ABB RobotStudio station: change_path.rspag

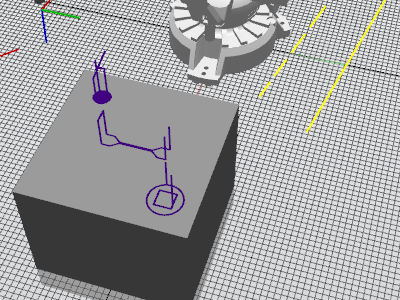
--- station ---
Station themal simulation (saved by RobotStudio 25.1.11133.0)
Controller IRB2600_12_185
  mechanical unit ROB_1: IRB2600_12_185__02, 6 joints, base frame (0, 0, 0) mm
Layout (positions relative to the parent item):
  - IRB2600_12_185__02 [mechanism, from %ABB.RobotStudio.Models.IRB2600%\IRB2600_12_185_G_02.rslib] at (0, 0, 0) mm; joint values [0, 0, 0, 0, 0.5236, 0] (rad or m)
  - AW_Gun_PSF_25 [mechanism, from %ABB.RobotStudio.Models.ArcWelding%\AW_Gun_PSF_25.rslib] at (1018.61, 0, 1417.5) mm, rotated rx 180 ry 60 rz 180 deg
  - Part_1 [part] at (100, 0, -100) mm, size 500 x 500 x 500 mm
Attachment: AW_Gun_PSF_25 is attached to IRB2600_12_185__02 / Link6

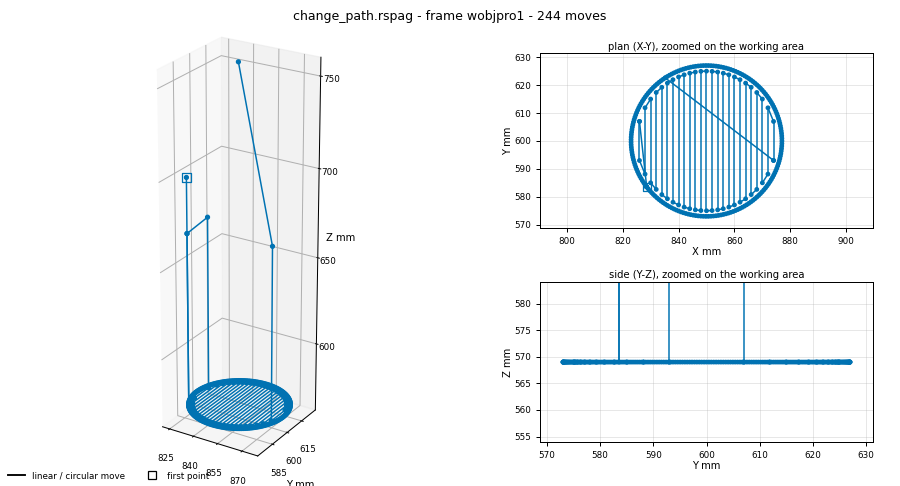
[picture p0: tool path of change_path.rspag in frame wobjpro1, 244 of 529 moves have a stored position in this frame; points joined in program order, loops and branches not executed]
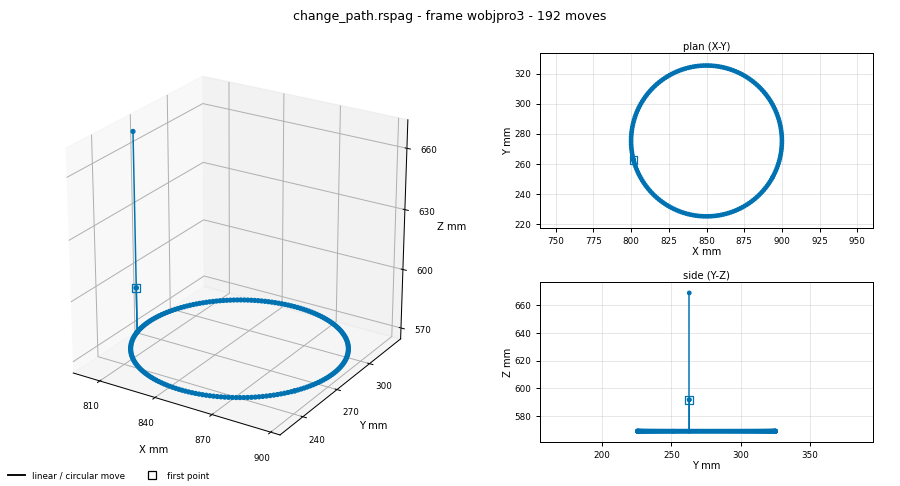
[picture p1: tool path of change_path.rspag in frame wobjpro3, 192 of 529 moves have a stored position in this frame; points joined in program order, loops and branches not executed]
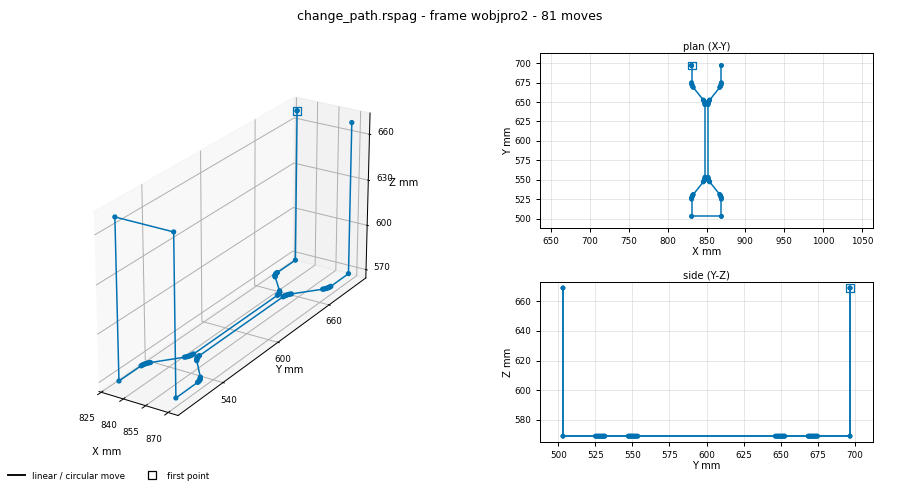
[picture p2: tool path of change_path.rspag in frame wobjpro2, 81 of 529 moves have a stored position in this frame; points joined in program order, loops and branches not executed]
--- Controller Data/IRB2600_12_185/RAPID/TASK1/PROGMOD/CalibData.mod ---
MODULE CalibData
    PERS tooldata AW_Gun:=[TRUE,[[119.5,0,352],[0.890213743,0,0.455543074,0]],[1,[0,0,100],[1,0,0,0],0,0,0]];
    PERS tooldata tFronius:=[TRUE,[[119.5,0,352],[0.890213743,0,0.455543074,0]],[1,[0,0,100],[1,0,0,0],0,0,0]];
     TASK PERS wobjdata wobjpro1:=[FALSE,TRUE,"",[[-52.352266096,-751.940840166,-168.793042727],[1,0,0,0]],[[0,0,0.0541992],[1,0,0,0]]];
  TASK PERS wobjdata wobjpro2:=[FALSE,TRUE,"",[[101.173073889,-585.583883348,-168],[1,0,0,0]],[[0,0,-0.0836792],[1,0,0,0]]];
  TASK PERS wobjdata wobjpro3:=[FALSE,TRUE,"",[[251.773303947,-119.398296432,-164.096623534],[1,0,0,0]],[[0,0,-4.67993],[1,0,0,0]]];
   TASK PERS wobjdata wobjpro4:=[FALSE,TRUE,"",[[250.933389795,-444.202986893,-163.664818503],[1,0,0,0]],[[0,0,-5.12018],[1,0,0,0]]];
  TASK PERS wobjdata wobjcam:=[FALSE,TRUE,"",[[1100,380,580],[1,0,0,0]],[[0,0,0],[1,0,0,0]]];
  TASK PERS wobjdata dedicate_wobj:=[FALSE,TRUE,"",[[1003,385,578.53],[1,0,0,0]],[[0,0,11.1832],[1,0,0,0]]];


PERS tooldata Processhead1 := [TRUE,[[-1.72,-0.76,490.02],[-0.01344,-0.95371,-0.07753,0.29025]],[3,[1,0,300],[1,0,0,0],0,0,0]];


!! ************************************************************
!! Toolpath ID: 1724238657_MX3D8v7kg | MX3D
!! Chunk ID: 0 [1/1]
!! Robot: hv_waam cell
!! Filename: MX3D_20240821_151151.mod
!! Project name: MX3D
!! Created on 2024-08-21 15:11:51.971757
!! ************************************************************

!! Delays for 2mm layer strategy (Single Wall Contour):
VAR num delayClosedStart_0  := 0.05;
VAR num delayClosedStop_0   := 0.05;
VAR num delayOpenStart_0    := 0.25;
VAR num delayOpenStop_0     := 0.1;


!! Delays for 2.6 mm layer strategy (Single Wall Contour):
VAR num delayClosedStart_1  := 0.05;
VAR num delayClosedStop_1   := 0.05;
VAR num delayOpenStart_1    := 0.1;
VAR num delayOpenStop_1     := 0.1;

VAR num delayOverhang       := 0;

!! Print and approach speeds
VAR speeddata printSpeed := [12, 500.0, 10.0, 10.0];
VAR speeddata moveSpeed := [800.0, 500.0, 300.0, 60.0];

!! Welding and process parameters
VAR bool useTempSensor    := TRUE;

VAR num wTime_25 := 25;
 CONST robtarget p30:=[[-49.36,-18.80,327.48],[0.761522,-0.0130271,0.0123584,0.647891],[0,1,-2,0],[9E+09,9E+09,9E+09,9E+09,9E+09,9E+09]];


VAR num wTime_5 := 5;

 !!PERS tooldata bendedTool:=[TRUE,[[-1.728,-0.7687,490.03],[0.0775305,-0.290248,-0.0134406,-0.953711]],[10,[85,0,65],[1,0,0,0],0.01,0.01,0.01]];
 PERS tooldata bendedTool:=[TRUE,[[119.5,0,352],[0.890213743,0,0.455543074,0]],[1,[0,0,100],[1,0,0,0],0,0,0]];
    TASK PERS wobjdata wobjWelding:=[FALSE,TRUE,"",[[700,-250,400],[1,0,0,0]],[[0,0,0],[1,0,0,0]]];
ENDMODULE

--- Controller Data/IRB2600_12_185/RAPID/TASK1/PROGMOD/Module1.mod ---
MODULE Module1
        CONST robtarget Target_10:=[[100,100,50],[0,0,1,0],[-1,1,-2,0],[9E+09,9E+09,9E+09,9E+09,9E+09,9E+09]];
    CONST robtarget Target_20:=[[100,400,50],[0,0,1,0],[0,2,-3,0],[9E+09,9E+09,9E+09,9E+09,9E+09,9E+09]];
    CONST robtarget Target_30:=[[400,400,50],[0,0,1,0],[0,2,-3,0],[9E+09,9E+09,9E+09,9E+09,9E+09,9E+09]];
    CONST robtarget Target_40:=[[400,100,50],[0,0,1,0],[-1,1,-2,0],[9E+09,9E+09,9E+09,9E+09,9E+09,9E+09]];
    CONST robtarget Target_50:=[[250,250,0],[0,0,1,0],[0,1,-2,0],[9E+09,9E+09,9E+09,9E+09,9E+09,9E+09]];
    CONST robtarget Target_10_1:=[[120,80,0],[0,0,1,0],[-1,1,-2,0],[9E+09,9E+09,9E+09,9E+09,9E+09,9E+09]];
    CONST robtarget Target_10_2:=[[80,80,0],[0,0,1,0],[-1,1,-2,0],[9E+09,9E+09,9E+09,9E+09,9E+09,9E+09]];
    CONST robtarget Target_10_3:=[[80,120,0],[0,0,1,0],[-1,1,-2,0],[9E+09,9E+09,9E+09,9E+09,9E+09,9E+09]];
    CONST robtarget Target_10_4:=[[120,120,0],[0,0,1,0],[-1,1,-2,0],[9E+09,9E+09,9E+09,9E+09,9E+09,9E+09]];
    CONST robtarget Target_20_1:=[[120,380,0],[0,0,1,0],[0,2,-3,0],[9E+09,9E+09,9E+09,9E+09,9E+09,9E+09]];
    CONST robtarget Target_20_2:=[[80,380,0],[0,0,1,0],[0,2,-3,0],[9E+09,9E+09,9E+09,9E+09,9E+09,9E+09]];
    CONST robtarget Target_20_3:=[[80,420,0],[0,0,1,0],[0,2,-3,0],[9E+09,9E+09,9E+09,9E+09,9E+09,9E+09]];
    CONST robtarget Target_20_4:=[[120,420,0],[0,0,1,0],[0,2,-3,0],[9E+09,9E+09,9E+09,9E+09,9E+09,9E+09]];
    CONST robtarget Target_30_1:=[[420,380,0],[0,0,1,0],[0,2,-3,0],[9E+09,9E+09,9E+09,9E+09,9E+09,9E+09]];
    CONST robtarget Target_30_2:=[[380,380,0],[0,0,1,0],[0,2,-3,0],[9E+09,9E+09,9E+09,9E+09,9E+09,9E+09]];
    CONST robtarget Target_30_3:=[[380,420,0],[0,0,1,0],[0,2,-3,0],[9E+09,9E+09,9E+09,9E+09,9E+09,9E+09]];
    CONST robtarget Target_30_4:=[[420,420,0],[0,0,1,0],[0,2,-3,0],[9E+09,9E+09,9E+09,9E+09,9E+09,9E+09]];
    CONST robtarget Target_40_1:=[[420,80,0],[0,0,1,0],[-1,1,-2,0],[9E+09,9E+09,9E+09,9E+09,9E+09,9E+09]];
    CONST robtarget Target_40_2:=[[380,80,0],[0,0,1,0],[-1,1,-2,0],[9E+09,9E+09,9E+09,9E+09,9E+09,9E+09]];
    CONST robtarget Target_40_3:=[[380,120,0],[0,0,1,0],[-1,1,-2,0],[9E+09,9E+09,9E+09,9E+09,9E+09,9E+09]];
    CONST robtarget Target_40_4:=[[420,120,0],[0,0,1,0],[-1,1,-2,0],[9E+09,9E+09,9E+09,9E+09,9E+09,9E+09]];
    VAR num interpassTemp;
    VAR num emissivity;
    VAR num numtemp;


!***********************************************************
    !
    ! Module:  Module1
    !
    ! Description:
    !   <Insert description here>
    !
    ! Author: xizh0002
    !
    ! Version: 1.0
    !
    !***********************************************************


    !***********************************************************
    !
    ! Procedure main
    !
    !   This is the entry point of your program
    !
    !***********************************************************
    PROC main()
        tempmeas;
    ENDPROC

    PROC tempmeas()
        r_cutwire;
    	MoveJ [[-130.39,-18.86,150.5],[0.0697509,0.000014922,-0.000044012,-0.997564],[0,-1,0,0],[9E+09,9E+09,9E+09,9E+09,9E+09,9E+09]],v500,z50,bendedTool\WObj:=wobjcam;
    	MoveJ [[31.69,367.16,1210],[0.276174,0.456891,0.112412,-0.838058],[0,0,-1,0],[9E+09,9E+09,9E+09,9E+09,9E+09,9E+09]],v800,z50,bendedTool\WObj:=wobjcam;
        tpreadfk reg1,"What to print?", "dia100","square","fork","solid","SKIP";
        MoveL [[-8.44,117.89,200],[0.0697498,-0.00001779,-0.00000352,-0.997564],[0,-1,0,0],[9E+09,9E+09,9E+09,9E+09,9E+09,9E+09]],v500,z50,bendedTool\WObj:=wobjcam;
        IF reg1=1 THEN
            dia100;
        ENDIF

        IF reg1=2 THEN
            square;
        ENDIF

        IF reg1=3 THEN
            gaffel;
        ENDIF

        IF reg1=4 THEN
            solid;
        ENDIF
    ENDPROC


PROC solid()
VAR robtarget touchpoint:=[[824.662,609.333,565],[0.000000,0.997564,0.069756,0.000000],[0,-1,0,0],[9E9,9E9,9E9,9E9,9E9,9E9]];
interpassTemp := 200.0;
emissivity := 0.992;
MoveL [[828.586,583.552,700],[0,0.997564,0.069756,0],[0,-1,0,0],[9E+09,9E+09,9E+09,9E+09,9E+09,9E+09]],moveSpeed,z0,bendedTool\WObj:=wobjpro1;
serch_height 0,0,touchpoint,numtemp;
!(num ofx, num ofy, robtarget target, inout num zval)
wobjpro1.oframe.trans.z:=numtemp-569.010;



MoveL [[828.586,583.552,669],[0,0.997564,0.069756,0],[0,-1,0,0],[9E+09,9E+09,9E+09,9E+09,9E+09,9E+09]],moveSpeed,z0,bendedTool\WObj:=wobjpro1;
MoveL [[828.586,583.552,569.01],[0,0.997564,0.069756,0],[0,-1,0,0],[9E+09,9E+09,9E+09,9E+09,9E+09,9E+09]],moveSpeed,fine,bendedTool\WObj:=wobjpro1;

startcontinuousweld; !layer  \delay:=delayClosedStart_0 \weldingProgram:=3 \weldId:="0000-0000-0000-0002";
TPWrite "[0.5%] PRT0 LYR0 TRK0 (700.0mm)";
MoveL [[828.048,584.277,569.01],[0,0.997564,0.069756,0],[0,-1,0,0],[9E+09,9E+09,9E+09,9E+09,9E+09,9E+09]],printSpeed,z0,bendedTool\WObj:=wobjpro1;
MoveL [[827.532,585.023,569.01],[0,0.997564,0.069756,0],[0,-1,0,0],[9E+09,9E+09,9E+09,9E+09,9E+09,9E+09]],printSpeed,z0,bendedTool\WObj:=wobjpro1;
MoveL [[827.042,585.786,569.01],[0,0.997564,0.069756,0],[0,-1,0,0],[9E+09,9E+09,9E+09,9E+09,9E+09,9E+09]],printSpeed,z0,bendedTool\WObj:=wobjpro1;
MoveL [[826.575,586.569,569.01],[0,0.997564,0.069756,0],[0,-1,0,0],[9E+09,9E+09,9E+09,9E+09,9E+09,9E+09]],printSpeed,z0,bendedTool\WObj:=wobjpro1;
MoveL [[826.139,587.36,569.01],[0,0.997564,0.069756,0],[0,-1,0,0],[9E+09,9E+09,9E+09,9E+09,9E+09,9E+09]],printSpeed,z0,bendedTool\WObj:=wobjpro1;
MoveL [[825.728,588.168,569.01],[0,0.997564,0.069756,0],[0,-1,0,0],[9E+09,9E+09,9E+09,9E+09,9E+09,9E+09]],printSpeed,z0,bendedTool\WObj:=wobjpro1;
MoveL [[825.344,588.99,569.01],[0,0.997564,0.069756,0],[0,-1,0,0],[9E+09,9E+09,9E+09,9E+09,9E+09,9E+09]],printSpeed,z0,bendedTool\WObj:=wobjpro1;
MoveL [[824.988,589.825,569.01],[0,0.997564,0.069756,0],[0,-1,0,0],[9E+09,9E+09,9E+09,9E+09,9E+09,9E+09]],printSpeed,z0,bendedTool\WObj:=wobjpro1;
MoveL [[824.661,590.671,569.01],[0,0.997564,0.069756,0],[0,-1,0,0],[9E+09,9E+09,9E+09,9E+09,9E+09,9E+09]],printSpeed,z0,bendedTool\WObj:=wobjpro1;
MoveL [[824.362,591.527,569.01],[0,0.997564,0.069756,0],[0,-1,0,0],[9E+09,9E+09,9E+09,9E+09,9E+09,9E+09]],printSpeed,z0,bendedTool\WObj:=wobjpro1;
MoveL [[824.091,592.393,569.01],[0,0.997564,0.069756,0],[0,-1,0,0],[9E+09,9E+09,9E+09,9E+09,9E+09,9E+09]],printSpeed,z0,bendedTool\WObj:=wobjpro1;
MoveL [[823.849,593.272,569.01],[0,0.997564,0.069756,0],[0,-1,0,0],[9E+09,9E+09,9E+09,9E+09,9E+09,9E+09]],printSpeed,z0,bendedTool\WObj:=wobjpro1;
MoveL [[823.639,594.15,569.01],[0,0.997564,0.069756,0],[0,-1,0,0],[9E+09,9E+09,9E+09,9E+09,9E+09,9E+09]],printSpeed,z0,bendedTool\WObj:=wobjpro1;
MoveL [[823.457,595.039,569.01],[0,0.997564,0.069756,0],[0,-1,0,0],[9E+09,9E+09,9E+09,9E+09,9E+09,9E+09]],printSpeed,z0,bendedTool\WObj:=wobjpro1;
MoveL [[823.306,595.933,569.01],[0,0.997564,0.069756,0],[0,-1,0,0],[9E+09,9E+09,9E+09,9E+09,9E+09,9E+09]],printSpeed,z0,bendedTool\WObj:=wobjpro1;
MoveL [[823.184,596.836,569.01],[0,0.997564,0.069756,0],[0,-1,0,0],[9E+09,9E+09,9E+09,9E+09,9E+09,9E+09]],printSpeed,z0,bendedTool\WObj:=wobjpro1;
MoveL [[823.093,597.735,569.01],[0,0.997564,0.069756,0],[0,-1,0,0],[9E+09,9E+09,9E+09,9E+09,9E+09,9E+09]],printSpeed,z0,bendedTool\WObj:=wobjpro1;
MoveL [[823.032,598.644,569.01],[0,0.997564,0.069756,0],[0,-1,0,0],[9E+09,9E+09,9E+09,9E+09,9E+09,9E+09]],printSpeed,z0,bendedTool\WObj:=wobjpro1;
MoveL [[823.002,599.551,569.01],[0,0.997564,0.069756,0],[0,-1,0,0],[9E+09,9E+09,9E+09,9E+09,9E+09,9E+09]],printSpeed,z0,bendedTool\WObj:=wobjpro1;
MoveL [[823.002,600.454,569.01],[0,0.997564,0.069756,0],[0,-1,0,0],[9E+09,9E+09,9E+09,9E+09,9E+09,9E+09]],printSpeed,z0,bendedTool\WObj:=wobjpro1;
MoveL [[823.032,601.36,569.01],[0,0.997564,0.069756,0],[0,-1,0,0],[9E+09,9E+09,9E+09,9E+09,9E+09,9E+09]],printSpeed,z0,bendedTool\WObj:=wobjpro1;
MoveL [[823.093,602.265,569.01],[0,0.997564,0.069756,0],[0,-1,0,0],[9E+09,9E+09,9E+09,9E+09,9E+09,9E+09]],printSpeed,z0,bendedTool\WObj:=wobjpro1;
MoveL [[823.184,603.168,569.01],[0,0.997564,0.069756,0],[0,-1,0,0],[9E+09,9E+09,9E+09,9E+09,9E+09,9E+09]],printSpeed,z0,bendedTool\WObj:=wobjpro1;
MoveL [[823.306,604.071,569.01],[0,0.997564,0.069756,0],[0,-1,0,0],[9E+09,9E+09,9E+09,9E+09,9E+09,9E+09]],printSpeed,z0,bendedTool\WObj:=wobjpro1;
MoveL [[823.457,604.961,569.01],[0,0.997564,0.069756,0],[0,-1,0,0],[9E+09,9E+09,9E+09,9E+09,9E+09,9E+09]],printSpeed,z0,bendedTool\WObj:=wobjpro1;
MoveL [[823.639,605.85,569.01],[0,0.997564,0.069756,0],[0,-1,0,0],[9E+09,9E+09,9E+09,9E+09,9E+09,9E+09]],printSpeed,z0,bendedTool\WObj:=wobjpro1;
MoveL [[823.85,606.732,569.01],[0,0.997564,0.069756,0],[0,-1,0,0],[9E+09,9E+09,9E+09,9E+09,9E+09,9E+09]],printSpeed,z0,bendedTool\WObj:=wobjpro1;
MoveL [[824.091,607.607,569.01],[0,0.997564,0.069756,0],[0,-1,0,0],[9E+09,9E+09,9E+09,9E+09,9E+09,9E+09]],printSpeed,z0,bendedTool\WObj:=wobjpro1;
MoveL [[824.363,608.477,569.01],[0,0.997564,0.069756,0],[0,-1,0,0],[9E+09,9E+09,9E+09,9E+09,9E+09,9E+09]],printSpeed,z0,bendedTool\WObj:=wobjpro1;
MoveL [[824.662,609.333,569.01],[0,0.997564,0.069756,0],[0,-1,0,0],[9E+09,9E+09,9E+09,9E+09,9E+09,9E+09]],printSpeed,z0,bendedTool\WObj:=wobjpro1;
MoveL [[824.988,610.175,569.01],[0,0.997564,0.069756,0],[0,-1,0,0],[9E+09,9E+09,9E+09,9E+09,9E+09,9E+09]],printSpeed,z0,bendedTool\WObj:=wobjpro1;
MoveL [[825.344,611.01,569.01],[0,0.997564,0.069756,0],[0,-1,0,0],[9E+09,9E+09,9E+09,9E+09,9E+09,9E+09]],printSpeed,z0,bendedTool\WObj:=wobjpro1;
MoveL [[825.73,611.836,569.01],[0,0.997564,0.069756,0],[0,-1,0,0],[9E+09,9E+09,9E+09,9E+09,9E+09,9E+09]],printSpeed,z0,bendedTool\WObj:=wobjpro1;
MoveL [[826.139,612.64,569.01],[0,0.997564,0.069756,0],[0,-1,0,0],[9E+09,9E+09,9E+09,9E+09,9E+09,9E+09]],printSpeed,z0,bendedTool\WObj:=wobjpro1;
MoveL [[826.577,613.435,569.01],[0,0.997564,0.069756,0],[0,-1,0,0],[9E+09,9E+09,9E+09,9E+09,9E+09,9E+09]],printSpeed,z0,bendedTool\WObj:=wobjpro1;
MoveL [[827.044,614.218,569.01],[0,0.997564,0.069756,0],[0,-1,0,0],[9E+09,9E+09,9E+09,9E+09,9E+09,9E+09]],printSpeed,z0,bendedTool\WObj:=wobjpro1;
MoveL [[827.535,614.981,569.01],[0,0.997564,0.069756,0],[0,-1,0,0],[9E+09,9E+09,9E+09,9E+09,9E+09,9E+09]],printSpeed,z0,bendedTool\WObj:=wobjpro1;
MoveL [[828.048,615.723,569.01],[0,0.997564,0.069756,0],[0,-1,0,0],[9E+09,9E+09,9E+09,9E+09,9E+09,9E+09]],printSpeed,z0,bendedTool\WObj:=wobjpro1;
MoveL [[828.589,616.452,569.01],[0,0.997564,0.069756,0],[0,-1,0,0],[9E+09,9E+09,9E+09,9E+09,9E+09,9E+09]],printSpeed,z0,bendedTool\WObj:=wobjpro1;
MoveL [[829.156,617.165,569.01],[0,0.997564,0.069756,0],[0,-1,0,0],[9E+09,9E+09,9E+09,9E+09,9E+09,9E+09]],printSpeed,z0,bendedTool\WObj:=wobjpro1;
MoveL [[829.742,617.852,569.01],[0,0.997564,0.069756,0],[0,-1,0,0],[9E+09,9E+09,9E+09,9E+09,9E+09,9E+09]],printSpeed,z0,bendedTool\WObj:=wobjpro1;
MoveL [[830.356,618.526,569.01],[0,0.997564,0.069756,0],[0,-1,0,0],[9E+09,9E+09,9E+09,9E+09,9E+09,9E+09]],printSpeed,z0,bendedTool\WObj:=wobjpro1;
MoveL [[830.986,619.172,569.01],[0,0.997564,0.069756,0],[0,-1,0,0],[9E+09,9E+09,9E+09,9E+09,9E+09,9E+09]],printSpeed,z0,bendedTool\WObj:=wobjpro1;
MoveL [[831.641,619.8,569.01],[0,0.997564,0.069756,0],[0,-1,0,0],[9E+09,9E+09,9E+09,9E+09,9E+09,9E+09]],printSpeed,z0,bendedTool\WObj:=wobjpro1;
MoveL [[832.317,620.405,569.01],[0,0.997564,0.069756,0],[0,-1,0,0],[9E+09,9E+09,9E+09,9E+09,9E+09,9E+09]],printSpeed,z0,bendedTool\WObj:=wobjpro1;
MoveL [[833.012,620.988,569.01],[0,0.997564,0.069756,0],[0,-1,0,0],[9E+09,9E+09,9E+09,9E+09,9E+09,9E+09]],printSpeed,z0,bendedTool\WObj:=wobjpro1;
MoveL [[833.727,621.547,569.01],[0,0.997564,0.069756,0],[0,-1,0,0],[9E+09,9E+09,9E+09,9E+09,9E+09,9E+09]],printSpeed,z0,bendedTool\WObj:=wobjpro1;
MoveL [[834.46,622.081,569.01],[0,0.997564,0.069756,0],[0,-1,0,0],[9E+09,9E+09,9E+09,9E+09,9E+09,9E+09]],printSpeed,z0,bendedTool\WObj:=wobjpro1;
MoveL [[835.21,622.591,569.01],[0,0.997564,0.069756,0],[0,-1,0,0],[9E+09,9E+09,9E+09,9E+09,9E+09,9E+09]],printSpeed,z0,bendedTool\WObj:=wobjpro1;
MoveL [[835.978,623.075,569.01],[0,0.997564,0.069756,0],[0,-1,0,0],[9E+09,9E+09,9E+09,9E+09,9E+09,9E+09]],printSpeed,z0,bendedTool\WObj:=wobjpro1;
MoveL [[836.761,623.533,569.01],[0,0.997564,0.069756,0],[0,-1,0,0],[9E+09,9E+09,9E+09,9E+09,9E+09,9E+09]],printSpeed,z0,bendedTool\WObj:=wobjpro1;
MoveL [[837.563,623.966,569.01],[0,0.997564,0.069756,0],[0,-1,0,0],[9E+09,9E+09,9E+09,9E+09,9E+09,9E+09]],printSpeed,z0,bendedTool\WObj:=wobjpro1;
MoveL [[838.371,624.368,569.01],[0,0.997564,0.069756,0],[0,-1,0,0],[9E+09,9E+09,9E+09,9E+09,9E+09,9E+09]],printSpeed,z0,bendedTool\WObj:=wobjpro1;
MoveL [[839.196,624.745,569.01],[0,0.997564,0.069756,0],[0,-1,0,0],[9E+09,9E+09,9E+09,9E+09,9E+09,9E+09]],printSpeed,z0,bendedTool\WObj:=wobjpro1;
MoveL [[840.033,625.094,569.01],[0,0.997564,0.069756,0],[0,-1,0,0],[9E+09,9E+09,9E+09,9E+09,9E+09,9E+09]],printSpeed,z0,bendedTool\WObj:=wobjpro1;
MoveL [[840.886,625.416,569.01],[0,0.997564,0.069756,0],[0,-1,0,0],[9E+09,9E+09,9E+09,9E+09,9E+09,9E+09]],printSpeed,z0,bendedTool\WObj:=wobjpro1;
MoveL [[841.741,625.707,569.01],[0,0.997564,0.069756,0],[0,-1,0,0],[9E+09,9E+09,9E+09,9E+09,9E+09,9E+09]],printSpeed,z0,bendedTool\WObj:=wobjpro1;
MoveL [[842.609,625.97,569.01],[0,0.997564,0.069756,0],[0,-1,0,0],[9E+09,9E+09,9E+09,9E+09,9E+09,9E+09]],printSpeed,z0,bendedTool\WObj:=wobjpro1;
MoveL [[843.49,626.204,569.01],[0,0.997564,0.069756,0],[0,-1,0,0],[9E+09,9E+09,9E+09,9E+09,9E+09,9E+09]],printSpeed,z0,bendedTool\WObj:=wobjpro1;
MoveL [[844.37,626.407,569.01],[0,0.997564,0.069756,0],[0,-1,0,0],[9E+09,9E+09,9E+09,9E+09,9E+09,9E+09]],printSpeed,z0,bendedTool\WObj:=wobjpro1;
MoveL [[845.264,626.582,569.01],[0,0.997564,0.069756,0],[0,-1,0,0],[9E+09,9E+09,9E+09,9E+09,9E+09,9E+09]],printSpeed,z0,bendedTool\WObj:=wobjpro1;
MoveL [[846.155,626.725,569.01],[0,0.997564,0.069756,0],[0,-1,0,0],[9E+09,9E+09,9E+09,9E+09,9E+09,9E+09]],printSpeed,z0,bendedTool\WObj:=wobjpro1;
MoveL [[847.055,626.839,569.01],[0,0.997564,0.069756,0],[0,-1,0,0],[9E+09,9E+09,9E+09,9E+09,9E+09,9E+09]],printSpeed,z0,bendedTool\WObj:=wobjpro1;
MoveL [[847.959,626.923,569.01],[0,0.997564,0.069756,0],[0,-1,0,0],[9E+09,9E+09,9E+09,9E+09,9E+09,9E+09]],printSpeed,z0,bendedTool\WObj:=wobjpro1;
MoveL [[848.864,626.976,569.01],[0,0.997564,0.069756,0],[0,-1,0,0],[9E+09,9E+09,9E+09,9E+09,9E+09,9E+09]],printSpeed,z0,bendedTool\WObj:=wobjpro1;
MoveL [[849.776,626.999,569.01],[0,0.997564,0.069756,0],[0,-1,0,0],[9E+09,9E+09,9E+09,9E+09,9E+09,9E+09]],printSpeed,z0,bendedTool\WObj:=wobjpro1;
MoveL [[850.679,626.992,569.01],[0,0.997564,0.069756,0],[0,-1,0,0],[9E+09,9E+09,9E+09,9E+09,9E+09,9E+09]],printSpeed,z0,bendedTool\WObj:=wobjpro1;
MoveL [[851.589,626.953,569.01],[0,0.997564,0.069756,0],[0,-1,0,0],[9E+09,9E+09,9E+09,9E+09,9E+09,9E+09]],printSpeed,z0,bendedTool\WObj:=wobjpro1;
MoveL [[852.489,626.885,569.01],[0,0.997564,0.069756,0],[0,-1,0,0],[9E+09,9E+09,9E+09,9E+09,9E+09,9E+09]],printSpeed,z0,bendedTool\WObj:=wobjpro1;
MoveL [[853.395,626.786,569.01],[0,0.997564,0.069756,0],[0,-1,0,0],[9E+09,9E+09,9E+09,9E+09,9E+09,9E+09]],printSpeed,z0,bendedTool\WObj:=wobjpro1;
MoveL [[854.289,626.657,569.01],[0,0.997564,0.069756,0],[0,-1,0,0],[9E+09,9E+09,9E+09,9E+09,9E+09,9E+09]],printSpeed,z0,bendedTool\WObj:=wobjpro1;
MoveL [[855.186,626.497,569.01],[0,0.997564,0.069756,0],[0,-1,0,0],[9E+09,9E+09,9E+09,9E+09,9E+09,9E+09]],printSpeed,z0,bendedTool\WObj:=wobjpro1;
MoveL [[856.069,626.309,569.01],[0,0.997564,0.069756,0],[0,-1,0,0],[9E+09,9E+09,9E+09,9E+09,9E+09,9E+09]],printSpeed,z0,bendedTool\WObj:=wobjpro1;
MoveL [[856.95,626.09,569.01],[0,0.997564,0.069756,0],[0,-1,0,0],[9E+09,9E+09,9E+09,9E+09,9E+09,9E+09]],printSpeed,z0,bendedTool\WObj:=wobjpro1;
MoveL [[857.822,625.842,569.01],[0,0.997564,0.069756,0],[0,-1,0,0],[9E+09,9E+09,9E+09,9E+09,9E+09,9E+09]],printSpeed,z0,bendedTool\WObj:=wobjpro1;
MoveL [[858.686,625.564,569.01],[0,0.997564,0.069756,0],[0,-1,0,0],[9E+09,9E+09,9E+09,9E+09,9E+09,9E+09]],printSpeed,z0,bendedTool\WObj:=wobjpro1;
MoveL [[859.54,625.258,569.01],[0,0.997564,0.069756,0],[0,-1,0,0],[9E+09,9E+09,9E+09,9E+09,9E+09,9E+09]],printSpeed,z0,bendedTool\WObj:=wobjpro1;
MoveL [[860.383,624.923,569.01],[0,0.997564,0.069756,0],[0,-1,0,0],[9E+09,9E+09,9E+09,9E+09,9E+09,9E+09]],printSpeed,z0,bendedTool\WObj:=wobjpro1;
MoveL [[861.214,624.56,569.01],[0,0.997564,0.069756,0],[0,-1,0,0],[9E+09,9E+09,9E+09,9E+09,9E+09,9E+09]],printSpeed,z0,bendedTool\WObj:=wobjpro1;
MoveL [[862.033,624.17,569.01],[0,0.997564,0.069756,0],[0,-1,0,0],[9E+09,9E+09,9E+09,9E+09,9E+09,9E+09]],printSpeed,z0,bendedTool\WObj:=wobjpro1;
MoveL [[862.842,623.75,569.01],[0,0.997564,0.069756,0],[0,-1,0,0],[9E+09,9E+09,9E+09,9E+09,9E+09,9E+09]],printSpeed,z0,bendedTool\WObj:=wobjpro1;
MoveL [[863.629,623.307,569.01],[0,0.997564,0.069756,0],[0,-1,0,0],[9E+09,9E+09,9E+09,9E+09,9E+09,9E+09]],printSpeed,z0,bendedTool\WObj:=wobjpro1;
MoveL [[864.408,622.833,569.01],[0,0.997564,0.069756,0],[0,-1,0,0],[9E+09,9E+09,9E+09,9E+09,9E+09,9E+09]],printSpeed,z0,bendedTool\WObj:=wobjpro1;
MoveL [[865.167,622.336,569.01],[0,0.997564,0.069756,0],[0,-1,0,0],[9E+09,9E+09,9E+09,9E+09,9E+09,9E+09]],printSpeed,z0,bendedTool\WObj:=wobjpro1;
MoveL [[865.909,621.814,569.01],[0,0.997564,0.069756,0],[0,-1,0,0],[9E+09,9E+09,9E+09,9E+09,9E+09,9E+09]],printSpeed,z0,bendedTool\WObj:=wobjpro1;
MoveL [[866.629,621.27,569.01],[0,0.997564,0.069756,0],[0,-1,0,0],[9E+09,9E+09,9E+09,9E+09,9E+09,9E+09]],printSpeed,z0,bendedTool\WObj:=wobjpro1;
MoveL [[867.334,620.7,569.01],[0,0.997564,0.069756,0],[0,-1,0,0],[9E+09,9E+09,9E+09,9E+09,9E+09,9E+09]],printSpeed,z0,bendedTool\WObj:=wobjpro1;
MoveL [[868.02,620.106,569.01],[0,0.997564,0.069756,0],[0,-1,0,0],[9E+09,9E+09,9E+09,9E+09,9E+09,9E+09]],printSpeed,z0,bendedTool\WObj:=wobjpro1;
MoveL [[868.688,619.486,569.01],[0,0.997564,0.069756,0],[0,-1,0,0],[9E+09,9E+09,9E+09,9E+09,9E+09,9E+09]],printSpeed,z0,bendedTool\WObj:=wobjpro1;
MoveL [[869.332,618.847,569.01],[0,0.997564,0.069756,0],[0,-1,0,0],[9E+09,9E+09,9E+09,9E+09,9E+09,9E+09]],printSpeed,z0,bendedTool\WObj:=wobjpro1;
MoveL [[869.951,618.19,569.01],[0,0.997564,0.069756,0],[0,-1,0,0],[9E+09,9E+09,9E+09,9E+09,9E+09,9E+09]],printSpeed,z0,bendedTool\WObj:=wobjpro1;
MoveL [[870.554,617.506,569.01],[0,0.997564,0.069756,0],[0,-1,0,0],[9E+09,9E+09,9E+09,9E+09,9E+09,9E+09]],printSpeed,z0,bendedTool\WObj:=wobjpro1;
MoveL [[871.128,616.809,569.01],[0,0.997564,0.069756,0],[0,-1,0,0],[9E+09,9E+09,9E+09,9E+09,9E+09,9E+09]],printSpeed,z0,bendedTool\WObj:=wobjpro1;
MoveL [[871.681,616.09,569.01],[0,0.997564,0.069756,0],[0,-1,0,0],[9E+09,9E+09,9E+09,9E+09,9E+09,9E+09]],printSpeed,z0,bendedTool\WObj:=wobjpro1;
MoveL [[872.209,615.352,569.01],[0,0.997564,0.069756,0],[0,-1,0,0],[9E+09,9E+09,9E+09,9E+09,9E+09,9E+09]],printSpeed,z0,bendedTool\WObj:=wobjpro1;
MoveL [[872.712,614.597,569.01],[0,0.997564,0.069756,0],[0,-1,0,0],[9E+09,9E+09,9E+09,9E+09,9E+09,9E+09]],printSpeed,z0,bendedTool\WObj:=wobjpro1;
MoveL [[873.19,613.826,569.01],[0,0.997564,0.069756,0],[0,-1,0,0],[9E+09,9E+09,9E+09,9E+09,9E+09,9E+09]],printSpeed,z0,bendedTool\WObj:=wobjpro1;
MoveL [[873.641,613.039,569.01],[0,0.997564,0.069756,0],[0,-1,0,0],[9E+09,9E+09,9E+09,9E+09,9E+09,9E+09]],printSpeed,z0,bendedTool\WObj:=wobjpro1;
MoveL [[874.068,612.234,569.01],[0,0.997564,0.069756,0],[0,-1,0,0],[9E+09,9E+09,9E+09,9E+09,9E+09,9E+09]],printSpeed,z0,bendedTool\WObj:=wobjpro1;
MoveL [[874.463,611.422,569.01],[0,0.997564,0.069756,0],[0,-1,0,0],[9E+09,9E+09,9E+09,9E+09,9E+09,9E+09]],printSpeed,z0,bendedTool\WObj:=wobjpro1;
MoveL [[874.833,610.594,569.01],[0,0.997564,0.069756,0],[0,-1,0,0],[9E+09,9E+09,9E+09,9E+09,9E+09,9E+09]],printSpeed,z0,bendedTool\WObj:=wobjpro1;
MoveL [[875.177,609.75,569.01],[0,0.997564,0.069756,0],[0,-1,0,0],[9E+09,9E+09,9E+09,9E+09,9E+09,9E+09]],printSpeed,z0,bendedTool\WObj:=wobjpro1;
MoveL [[875.488,608.902,569.01],[0,0.997564,0.069756,0],[0,-1,0,0],[9E+09,9E+09,9E+09,9E+09,9E+09,9E+09]],printSpeed,z0,bendedTool\WObj:=wobjpro1;
MoveL [[875.773,608.041,569.01],[0,0.997564,0.069756,0],[0,-1,0,0],[9E+09,9E+09,9E+09,9E+09,9E+09,9E+09]],printSpeed,z0,bendedTool\WObj:=wobjpro1;
MoveL [[876.029,607.171,569.01],[0,0.997564,0.069756,0],[0,-1,0,0],[9E+09,9E+09,9E+09,9E+09,9E+09,9E+09]],printSpeed,z0,bendedTool\WObj:=wobjpro1;
MoveL [[876.255,606.292,569.01],[0,0.997564,0.069756,0],[0,-1,0,0],[9E+09,9E+09,9E+09,9E+09,9E+09,9E+09]],printSpeed,z0,bendedTool\WObj:=wobjpro1;
MoveL [[876.451,605.406,569.01],[0,0.997564,0.069756,0],[0,-1,0,0],[9E+09,9E+09,9E+09,9E+09,9E+09,9E+09]],printSpeed,z0,bendedTool\WObj:=wobjpro1;
MoveL [[876.619,604.51,569.01],[0,0.997564,0.069756,0],[0,-1,0,0],[9E+09,9E+09,9E+09,9E+09,9E+09,9E+09]],printSpeed,z0,bendedTool\WObj:=wobjpro1;
MoveL [[876.755,603.618,569.01],[0,0.997564,0.069756,0],[0,-1,0,0],[9E+09,9E+09,9E+09,9E+09,9E+09,9E+09]],printSpeed,z0,bendedTool\WObj:=wobjpro1;
MoveL [[876.861,602.717,569.01],[0,0.997564,0.069756,0],[0,-1,0,0],[9E+09,9E+09,9E+09,9E+09,9E+09,9E+09]],printSpeed,z0,bendedTool\WObj:=wobjpro1;
MoveL [[876.937,601.813,569.01],[0,0.997564,0.069756,0],[0,-1,0,0],[9E+09,9E+09,9E+09,9E+09,9E+09,9E+09]],printSpeed,z0,bendedTool\WObj:=wobjpro1;
MoveL [[876.983,600.903,569.01],[0,0.997564,0.069756,0],[0,-1,0,0],[9E+09,9E+09,9E+09,9E+09,9E+09,9E+09]],printSpeed,z0,bendedTool\WObj:=wobjpro1;
MoveL [[876.998,599.995,569.01],[0,0.997564,0.069756,0],[0,-1,0,0],[9E+09,9E+09,9E+09,9E+09,9E+09,9E+09]],printSpeed,z0,bendedTool\WObj:=wobjpro1;
MoveL [[876.983,599.088,569.01],[0,0.997564,0.069756,0],[0,-1,0,0],[9E+09,9E+09,9E+09,9E+09,9E+09,9E+09]],printSpeed,z0,bendedTool\WObj:=wobjpro1;
MoveL [[876.937,598.182,569.01],[0,0.997564,0.069756,0],[0,-1,0,0],[9E+09,9E+09,9E+09,9E+09,9E+09,9E+09]],printSpeed,z0,bendedTool\WObj:=wobjpro1;
MoveL [[876.861,597.278,569.01],[0,0.997564,0.069756,0],[0,-1,0,0],[9E+09,9E+09,9E+09,9E+09,9E+09,9E+09]],printSpeed,z0,bendedTool\WObj:=wobjpro1;
MoveL [[876.754,596.378,569.01],[0,0.997564,0.069756,0],[0,-1,0,0],[9E+09,9E+09,9E+09,9E+09,9E+09,9E+09]],printSpeed,z0,bendedTool\WObj:=wobjpro1;
MoveL [[876.617,595.481,569.01],[0,0.997564,0.069756,0],[0,-1,0,0],[9E+09,9E+09,9E+09,9E+09,9E+09,9E+09]],printSpeed,z0,bendedTool\WObj:=wobjpro1;
MoveL [[876.45,594.589,569.01],[0,0.997564,0.069756,0],[0,-1,0,0],[9E+09,9E+09,9E+09,9E+09,9E+09,9E+09]],printSpeed,z0,bendedTool\WObj:=wobjpro1;
MoveL [[876.254,593.704,569.01],[0,0.997564,0.069756,0],[0,-1,0,0],[9E+09,9E+09,9E+09,9E+09,9E+09,9E+09]],printSpeed,z0,bendedTool\WObj:=wobjpro1;
MoveL [[876.027,592.825,569.01],[0,0.997564,0.069756,0],[0,-1,0,0],[9E+09,9E+09,9E+09,9E+09,9E+09,9E+09]],printSpeed,z0,bendedTool\WObj:=wobjpro1;
MoveL [[875.773,591.959,569.01],[0,0.997564,0.069756,0],[0,-1,0,0],[9E+09,9E+09,9E+09,9E+09,9E+09,9E+09]],printSpeed,z0,bendedTool\WObj:=wobjpro1;
MoveL [[875.488,591.098,569.01],[0,0.997564,0.069756,0],[0,-1,0,0],[9E+09,9E+09,9E+09,9E+09,9E+09,9E+09]],printSpeed,z0,bendedTool\WObj:=wobjpro1;
MoveL [[875.173,590.242,569.01],[0,0.997564,0.069756,0],[0,-1,0,0],[9E+09,9E+09,9E+09,9E+09,9E+09,9E+09]],printSpeed,z0,bendedTool\WObj:=wobjpro1;
MoveL [[874.833,589.406,569.01],[0,0.997564,0.069756,0],[0,-1,0,0],[9E+09,9E+09,9E+09,9E+09,9E+09,9E+09]],printSpeed,z0,bendedTool\WObj:=wobjpro1;
MoveL [[874.463,588.578,569.01],[0,0.997564,0.069756,0],[0,-1,0,0],[9E+09,9E+09,9E+09,9E+09,9E+09,9E+09]],printSpeed,z0,bendedTool\WObj:=wobjpro1;
MoveL [[874.064,587.758,569.01],[0,0.997564,0.069756,0],[0,-1,0,0],[9E+09,9E+09,9E+09,9E+09,9E+09,9E+09]],printSpeed,z0,bendedTool\WObj:=wobjpro1;
MoveL [[873.641,586.961,569.01],[0,0.997564,0.069756,0],[0,-1,0,0],[9E+09,9E+09,9E+09,9E+09,9E+09,9E+09]],printSpeed,z0,bendedTool\WObj:=wobjpro1;
MoveL [[873.19,586.174,569.01],[0,0.997564,0.069756,0],[0,-1,0,0],[9E+09,9E+09,9E+09,9E+09,9E+09,9E+09]],printSpeed,z0,bendedTool\WObj:=wobjpro1;
MoveL [[872.71,585.399,569.01],[0,0.997564,0.069756,0],[0,-1,0,0],[9E+09,9E+09,9E+09,9E+09,9E+09,9E+09]],printSpeed,z0,bendedTool\WObj:=wobjpro1;
MoveL [[872.209,584.648,569.01],[0,0.997564,0.069756,0],[0,-1,0,0],[9E+09,9E+09,9E+09,9E+09,9E+09,9E+09]],printSpeed,z0,bendedTool\WObj:=wobjpro1;
MoveL [[871.681,583.91,569.01],[0,0.997564,0.069756,0],[0,-1,0,0],[9E+09,9E+09,9E+09,9E+09,9E+09,9E+09]],printSpeed,z0,bendedTool\WObj:=wobjpro1;
MoveL [[871.128,583.191,569.01],[0,0.997564,0.069756,0],[0,-1,0,0],[9E+09,9E+09,9E+09,9E+09,9E+09,9E+09]],printSpeed,z0,bendedTool\WObj:=wobjpro1;
MoveL [[870.551,582.491,569.01],[0,0.997564,0.069756,0],[0,-1,0,0],[9E+09,9E+09,9E+09,9E+09,9E+09,9E+09]],printSpeed,z0,bendedTool\WObj:=wobjpro1;
MoveL [[869.951,581.81,569.01],[0,0.997564,0.069756,0],[0,-1,0,0],[9E+09,9E+09,9E+09,9E+09,9E+09,9E+09]],printSpeed,z0,bendedTool\WObj:=wobjpro1;
MoveL [[869.329,581.15,569.01],[0,0.997564,0.069756,0],[0,-1,0,0],[9E+09,9E+09,9E+09,9E+09,9E+09,9E+09]],printSpeed,z0,bendedTool\WObj:=wobjpro1;
MoveL [[868.685,580.511,569.01],[0,0.997564,0.069756,0],[0,-1,0,0],[9E+09,9E+09,9E+09,9E+09,9E+09,9E+09]],printSpeed,z0,bendedTool\WObj:=wobjpro1;
MoveL [[868.02,579.894,569.01],[0,0.997564,0.069756,0],[0,-1,0,0],[9E+09,9E+09,9E+09,9E+09,9E+09,9E+09]],printSpeed,z0,bendedTool\WObj:=wobjpro1;
MoveL [[867.331,579.298,569.01],[0,0.997564,0.069756,0],[0,-1,0,0],[9E+09,9E+09,9E+09,9E+09,9E+09,9E+09]],printSpeed,z0,bendedTool\WObj:=wobjpro1;
MoveL [[866.629,578.73,569.01],[0,0.997564,0.069756,0],[0,-1,0,0],[9E+09,9E+09,9E+09,9E+09,9E+09,9E+09]],printSpeed,z0,bendedTool\WObj:=wobjpro1;
MoveL [[865.905,578.183,569.01],[0,0.997564,0.069756,0],[0,-1,0,0],[9E+09,9E+09,9E+09,9E+09,9E+09,9E+09]],printSpeed,z0,bendedTool\WObj:=wobjpro1;
MoveL [[865.163,577.661,569.01],[0,0.997564,0.069756,0],[0,-1,0,0],[9E+09,9E+09,9E+09,9E+09,9E+09,9E+09]],printSpeed,z0,bendedTool\WObj:=wobjpro1;
MoveL [[864.404,577.164,569.01],[0,0.997564,0.069756,0],[0,-1,0,0],[9E+09,9E+09,9E+09,9E+09,9E+09,9E+09]],printSpeed,z0,bendedTool\WObj:=wobjpro1;
MoveL [[863.629,576.693,569.01],[0,0.997564,0.069756,0],[0,-1,0,0],[9E+09,9E+09,9E+09,9E+09,9E+09,9E+09]],printSpeed,z0,bendedTool\WObj:=wobjpro1;
MoveL [[862.838,576.248,569.01],[0,0.997564,0.069756,0],[0,-1,0,0],[9E+09,9E+09,9E+09,9E+09,9E+09,9E+09]],printSpeed,z0,bendedTool\WObj:=wobjpro1;
MoveL [[862.033,575.83,569.01],[0,0.997564,0.069756,0],[0,-1,0,0],[9E+09,9E+09,9E+09,9E+09,9E+09,9E+09]],printSpeed,z0,bendedTool\WObj:=wobjpro1;
MoveL [[861.21,575.438,569.01],[0,0.997564,0.069756,0],[0,-1,0,0],[9E+09,9E+09,9E+09,9E+09,9E+09,9E+09]],printSpeed,z0,bendedTool\WObj:=wobjpro1;
MoveL [[860.383,575.077,569.01],[0,0.997564,0.069756,0],[0,-1,0,0],[9E+09,9E+09,9E+09,9E+09,9E+09,9E+09]],printSpeed,z0,bendedTool\WObj:=wobjpro1;
MoveL [[859.54,574.742,569.01],[0,0.997564,0.069756,0],[0,-1,0,0],[9E+09,9E+09,9E+09,9E+09,9E+09,9E+09]],printSpeed,z0,bendedTool\WObj:=wobjpro1;
MoveL [[858.686,574.436,569.01],[0,0.997564,0.069756,0],[0,-1,0,0],[9E+09,9E+09,9E+09,9E+09,9E+09,9E+09]],printSpeed,z0,bendedTool\WObj:=wobjpro1;
MoveL [[857.822,574.158,569.01],[0,0.997564,0.069756,0],[0,-1,0,0],[9E+09,9E+09,9E+09,9E+09,9E+09,9E+09]],printSpeed,z0,bendedTool\WObj:=wobjpro1;
MoveL [[856.95,573.91,569.01],[0,0.997564,0.069756,0],[0,-1,0,0],[9E+09,9E+09,9E+09,9E+09,9E+09,9E+09]],printSpeed,z0,bendedTool\WObj:=wobjpro1;
MoveL [[856.069,573.691,569.01],[0,0.997564,0.069756,0],[0,-1,0,0],[9E+09,9E+09,9E+09,9E+09,9E+09,9E+09]],printSpeed,z0,bendedTool\WObj:=wobjpro1;
MoveL [[855.182,573.502,569.01],[0,0.997564,0.069756,0],[0,-1,0,0],[9E+09,9E+09,9E+09,9E+09,9E+09,9E+09]],printSpeed,z0,bendedTool\WObj:=wobjpro1;
MoveL [[854.289,573.343,569.01],[0,0.997564,0.069756,0],[0,-1,0,0],[9E+09,9E+09,9E+09,9E+09,9E+09,9E+09]],printSpeed,z0,bendedTool\WObj:=wobjpro1;
MoveL [[853.391,573.214,569.01],[0,0.997564,0.069756,0],[0,-1,0,0],[9E+09,9E+09,9E+09,9E+09,9E+09,9E+09]],printSpeed,z0,bendedTool\WObj:=wobjpro1;
MoveL [[852.485,573.115,569.01],[0,0.997564,0.069756,0],[0,-1,0,0],[9E+09,9E+09,9E+09,9E+09,9E+09,9E+09]],printSpeed,z0,bendedTool\WObj:=wobjpro1;
MoveL [[851.585,573.046,569.01],[0,0.997564,0.069756,0],[0,-1,0,0],[9E+09,9E+09,9E+09,9E+09,9E+09,9E+09]],printSpeed,z0,bendedTool\WObj:=wobjpro1;
MoveL [[850.678,573.008,569.01],[0,0.997564,0.069756,0],[0,-1,0,0],[9E+09,9E+09,9E+09,9E+09,9E+09,9E+09]],printSpeed,z0,bendedTool\WObj:=wobjpro1;
MoveL [[849.771,573.001,569.01],[0,0.997564,0.069756,0],[0,-1,0,0],[9E+09,9E+09,9E+09,9E+09,9E+09,9E+09]],printSpeed,z0,bendedTool\WObj:=wobjpro1;
MoveL [[848.864,573.024,569.01],[0,0.997564,0.069756,0],[0,-1,0,0],[9E+09,9E+09,9E+09,9E+09,9E+09,9E+09]],printSpeed,z0,bendedTool\WObj:=wobjpro1;
MoveL [[847.959,573.077,569.01],[0,0.997564,0.069756,0],[0,-1,0,0],[9E+09,9E+09,9E+09,9E+09,9E+09,9E+09]],printSpeed,z0,bendedTool\WObj:=wobjpro1;
MoveL [[847.055,573.161,569.01],[0,0.997564,0.069756,0],[0,-1,0,0],[9E+09,9E+09,9E+09,9E+09,9E+09,9E+09]],printSpeed,z0,bendedTool\WObj:=wobjpro1;
MoveL [[846.155,573.275,569.01],[0,0.997564,0.069756,0],[0,-1,0,0],[9E+09,9E+09,9E+09,9E+09,9E+09,9E+09]],printSpeed,z0,bendedTool\WObj:=wobjpro1;
MoveL [[845.256,573.42,569.01],[0,0.997564,0.069756,0],[0,-1,0,0],[9E+09,9E+09,9E+09,9E+09,9E+09,9E+09]],printSpeed,z0,bendedTool\WObj:=wobjpro1;
MoveL [[844.37,573.593,569.01],[0,0.997564,0.069756,0],[0,-1,0,0],[9E+09,9E+09,9E+09,9E+09,9E+09,9E+09]],printSpeed,z0,bendedTool\WObj:=wobjpro1;
MoveL [[843.486,573.797,569.01],[0,0.997564,0.069756,0],[0,-1,0,0],[9E+09,9E+09,9E+09,9E+09,9E+09,9E+09]],printSpeed,z0,bendedTool\WObj:=wobjpro1;
MoveL [[842.609,574.03,569.01],[0,0.997564,0.069756,0],[0,-1,0,0],[9E+09,9E+09,9E+09,9E+09,9E+09,9E+09]],printSpeed,z0,bendedTool\WObj:=wobjpro1;
MoveL [[841.741,574.293,569.01],[0,0.997564,0.069756,0],[0,-1,0,0],[9E+09,9E+09,9E+09,9E+09,9E+09,9E+09]],printSpeed,z0,bendedTool\WObj:=wobjpro1;
MoveL [[840.882,574.585,569.01],[0,0.997564,0.069756,0],[0,-1,0,0],[9E+09,9E+09,9E+09,9E+09,9E+09,9E+09]],printSpeed,z0,bendedTool\WObj:=wobjpro1;
MoveL [[840.033,574.906,569.01],[0,0.997564,0.069756,0],[0,-1,0,0],[9E+09,9E+09,9E+09,9E+09,9E+09,9E+09]],printSpeed,z0,bendedTool\WObj:=wobjpro1;
MoveL [[839.196,575.255,569.01],[0,0.997564,0.069756,0],[0,-1,0,0],[9E+09,9E+09,9E+09,9E+09,9E+09,9E+09]],printSpeed,z0,bendedTool\WObj:=wobjpro1;
MoveL [[838.371,575.632,569.01],[0,0.997564,0.069756,0],[0,-1,0,0],[9E+09,9E+09,9E+09,9E+09,9E+09,9E+09]],printSpeed,z0,bendedTool\WObj:=wobjpro1;
MoveL [[837.555,576.038,569.01],[0,0.997564,0.069756,0],[0,-1,0,0],[9E+09,9E+09,9E+09,9E+09,9E+09,9E+09]],printSpeed,z0,bendedTool\WObj:=wobjpro1;
MoveL [[836.757,576.47,569.01],[0,0.997564,0.069756,0],[0,-1,0,0],[9E+09,9E+09,9E+09,9E+09,9E+09,9E+09]],printSpeed,z0,bendedTool\WObj:=wobjpro1;
MoveL [[835.978,576.925,569.01],[0,0.997564,0.069756,0],[0,-1,0,0],[9E+09,9E+09,9E+09,9E+09,9E+09,9E+09]],printSpeed,z0,bendedTool\WObj:=wobjpro1;
MoveL [[835.21,577.409,569.01],[0,0.997564,0.069756,0],[0,-1,0,0],[9E+09,9E+09,9E+09,9E+09,9E+09,9E+09]],printSpeed,z0,bendedTool\WObj:=wobjpro1;
MoveL [[834.46,577.919,569.01],[0,0.997564,0.069756,0],[0,-1,0,0],[9E+09,9E+09,9E+09,9E+09,9E+09,9E+09]],printSpeed,z0,bendedTool\WObj:=wobjpro1;
MoveL [[833.727,578.453,569.01],[0,0.997564,0.069756,0],[0,-1,0,0],[9E+09,9E+09,9E+09,9E+09,9E+09,9E+09]],printSpeed,z0,bendedTool\WObj:=wobjpro1;
MoveL [[833.009,579.015,569.01],[0,0.997564,0.069756,0],[0,-1,0,0],[9E+09,9E+09,9E+09,9E+09,9E+09,9E+09]],printSpeed,z0,bendedTool\WObj:=wobjpro1;
MoveL [[832.317,579.595,569.01],[0,0.997564,0.069756,0],[0,-1,0,0],[9E+09,9E+09,9E+09,9E+09,9E+09,9E+09]],printSpeed,z0,bendedTool\WObj:=wobjpro1;
MoveL [[831.638,580.203,569.01],[0,0.997564,0.069756,0],[0,-1,0,0],[9E+09,9E+09,9E+09,9E+09,9E+09,9E+09]],printSpeed,z0,bendedTool\WObj:=wobjpro1;
MoveL [[830.986,580.828,569.01],[0,0.997564,0.069756,0],[0,-1,0,0],[9E+09,9E+09,9E+09,9E+09,9E+09,9E+09]],printSpeed,z0,bendedTool\WObj:=wobjpro1;
MoveL [[830.35,581.481,569.01],[0,0.997564,0.069756,0],[0,-1,0,0],[9E+09,9E+09,9E+09,9E+09,9E+09,9E+09]],printSpeed,z0,bendedTool\WObj:=wobjpro1;
MoveL [[829.742,582.148,569.01],[0,0.997564,0.069756,0],[0,-1,0,0],[9E+09,9E+09,9E+09,9E+09,9E+09,9E+09]],printSpeed,z0,bendedTool\WObj:=wobjpro1;
MoveL [[829.153,582.838,569.01],[0,0.997564,0.069756,0],[0,-1,0,0],[9E+09,9E+09,9E+09,9E+09,9E+09,9E+09]],printSpeed,z0,bendedTool\WObj:=wobjpro1;
MoveL [[828.586,583.552,569.01],[0,0.997564,0.069756,0],[0,-1,0,0],[9E+09,9E+09,9E+09,9E+09,9E+09,9E+09]],printSpeed,fine,bendedTool\WObj:=wobjpro1;
stopContinuousWeld \delay:=delayClosedStop_0;
MoveL [[828.586,583.552,669],[0,0.997564,0.069756,0],[0,-1,0,0],[9E+09,9E+09,9E+09,9E+09,9E+09,9E+09]],moveSpeed,z0,bendedTool\WObj:=wobjpro1;
MoveL [[826,607.005,669],[0,0.997564,0.069756,0],[0,-1,0,0],[9E+09,9E+09,9E+09,9E+09,9E+09,9E+09]],moveSpeed,z0,bendedTool\WObj:=wobjpro1;
MoveL [[826,607.005,569.01],[0,0.997564,0.069756,0],[0,-1,0,0],[9E+09,9E+09,9E+09,9E+09,9E+09,9E+09]],moveSpeed,fine,bendedTool\WObj:=wobjpro1;
printSpeed := [12.0, 500.0, 10.0, 10.0];
startcontinuousweld; !layer  \delay:=delayOpenStart_0 \weldingProgram:=3 \weldId:="0000-0000-0001-0002";
TPWrite "[43.2%] PRT0 LYR0 TRK1 (700.0mm)";
MoveL [[826,592.995,569.01],[0,0.997564,0.069756,0],[0,-1,0,0],[9E+09,9E+09,9E+09,9E+09,9E+09,9E+09]],printSpeed,fine,bendedTool\WObj:=wobjpro1;
!stopContinuousWeld \delay:=delayOpenStop_0;
!MoveL [[826.000,592.995,669],[0.000000,0.997564,0.069756,0.000000],[0,-1,0,0],[9E9,9E9,9E9,9E9,9E9,9E9]],moveSpeed,z0,bendedTool,\WObj:=wobjpro1;
!MoveL [[828.000,588.127,669],[0.000000,0.997564,0.069756,0.000000],[0,-1,0,0],[9E9,9E9,9E9,9E9,9E9,9E9]],moveSpeed,z0,bendedTool,\WObj:=wobjpro1;
MoveL [[828,588.127,569.01],[0,0.997564,0.069756,0],[0,-1,0,0],[9E+09,9E+09,9E+09,9E+09,9E+09,9E+09]],printSpeed,fine,bendedTool\WObj:=wobjpro1;
!startcontinuousweld; !layer  \delay:=delayOpenStart_0 \weldingProgram:=3 \weldId:="0000-0000-0002-0002";
TPWrite "[44.1%] PRT0 LYR0 TRK2 (700.0mm)";
MoveL [[828,611.873,569.01],[0,0.997564,0.069756,0],[0,-1,0,0],[9E+09,9E+09,9E+09,9E+09,9E+09,9E+09]],printSpeed,fine,bendedTool\WObj:=wobjpro1;
!stopContinuousWeld \delay:=delayOpenStop_0;
!MoveL [[828.000,611.873,669],[0.000000,0.997564,0.069756,0.000000],[0,-1,0,0],[9E9,9E9,9E9,9E9,9E9,9E9]],moveSpeed,z0,bendedTool,\WObj:=wobjpro1;
!MoveL [[830.000,614.997,669],[0.000000,0.997564,0.069756,0.000000],[0,-1,0,0],[9E9,9E9,9E9,9E9,9E9,9E9]],moveSpeed,z0,bendedTool,\WObj:=wobjpro1;
MoveL [[830,614.997,569.01],[0,0.997564,0.069756,0],[0,-1,0,0],[9E+09,9E+09,9E+09,9E+09,9E+09,9E+09]],printSpeed,fine,bendedTool\WObj:=wobjpro1;
!startcontinuousweld; !layer  \delay:=delayOpenStart_0 \weldingProgram:=3 \weldId:="0000-0000-0003-0002";
TPWrite "[45.0%] PRT0 LYR0 TRK3 (700.0mm)";
MoveL [[830,585.003,569.01],[0,0.997564,0.069756,0],[0,-1,0,0],[9E+09,9E+09,9E+09,9E+09,9E+09,9E+09]],printSpeed,fine,bendedTool\WObj:=wobjpro1;
!stopContinuousWeld \delay:=delayOpenStop_0;
!MoveL [[830.000,585.003,669],[0.000000,0.997564,0.069756,0.000000],[0,-1,0,0],[9E9,9E9,9E9,9E9,9E9,9E9]],moveSpeed,z0,bendedTool,\WObj:=wobjpro1;
!MoveL [[832.000,582.653,669],[0.000000,0.997564,0.069756,0.000000],[0,-1,0,0],[9E9,9E9,9E9,9E9,9E9,9E9]],moveSpeed,z0,bendedTool,\WObj:=wobjpro1;
MoveL [[832,582.653,569.01],[0,0.997564,0.069756,0],[0,-1,0,0],[9E+09,9E+09,9E+09,9E+09,9E+09,9E+09]],printSpeed,fine,bendedTool\WObj:=wobjpro1;
!startcontinuousweld; !layer  \delay:=delayOpenStart_0 \weldingProgram:=3 \weldId:="0000-0000-0004-0002";
TPWrite "[45.9%] PRT0 LYR0 TRK4 (700.0mm)";
MoveL [[832,617.347,569.01],[0,0.997564,0.069756,0],[0,-1,0,0],[9E+09,9E+09,9E+09,9E+09,9E+09,9E+09]],printSpeed,z0,bendedTool\WObj:=wobjpro1;
MoveL [[834,619.207,569.01],[0,0.997564,0.069756,0],[0,-1,0,0],[9E+09,9E+09,9E+09,9E+09,9E+09,9E+09]],printSpeed,z0,bendedTool\WObj:=wobjpro1;
MoveL [[834,580.793,569.01],[0,0.997564,0.069756,0],[0,-1,0,0],[9E+09,9E+09,9E+09,9E+09,9E+09,9E+09]],printSpeed,z0,bendedTool\WObj:=wobjpro1;
MoveL [[836,579.291,569.01],[0,0.997564,0.069756,0],[0,-1,0,0],[9E+09,9E+09,9E+09,9E+09,9E+09,9E+09]],printSpeed,z0,bendedTool\WObj:=wobjpro1;
MoveL [[836,620.709,569.01],[0,0.997564,0.069756,0],[0,-1,0,0],[9E+09,9E+09,9E+09,9E+09,9E+09,9E+09]],printSpeed,z0,bendedTool\WObj:=wobjpro1;
MoveL [[838,621.929,569.01],[0,0.997564,0.069756,0],[0,-1,0,0],[9E+09,9E+09,9E+09,9E+09,9E+09,9E+09]],printSpeed,z0,bendedTool\WObj:=wobjpro1;
MoveL [[838,578.071,569.01],[0,0.997564,0.069756,0],[0,-1,0,0],[9E+09,9E+09,9E+09,9E+09,9E+09,9E+09]],printSpeed,z0,bendedTool\WObj:=wobjpro1;
MoveL [[840,577.086,569.01],[0,0.997564,0.069756,0],[0,-1,0,0],[9E+09,9E+09,9E+09,9E+09,9E+09,9E+09]],printSpeed,z0,bendedTool\WObj:=wobjpro1;
MoveL [[840,622.914,569.01],[0,0.997564,0.069756,0],[0,-1,0,0],[9E+09,9E+09,9E+09,9E+09,9E+09,9E+09]],printSpeed,z0,bendedTool\WObj:=wobjpro1;
MoveL [[842,623.682,569.01],[0,0.997564,0.069756,0],[0,-1,0,0],[9E+09,9E+09,9E+09,9E+09,9E+09,9E+09]],printSpeed,z0,bendedTool\WObj:=wobjpro1;
MoveL [[842,576.318,569.01],[0,0.997564,0.069756,0],[0,-1,0,0],[9E+09,9E+09,9E+09,9E+09,9E+09,9E+09]],printSpeed,z0,bendedTool\WObj:=wobjpro1;
MoveL [[844,575.731,569.01],[0,0.997564,0.069756,0],[0,-1,0,0],[9E+09,9E+09,9E+09,9E+09,9E+09,9E+09]],printSpeed,z0,bendedTool\WObj:=wobjpro1;
MoveL [[844,624.269,569.01],[0,0.997564,0.069756,0],[0,-1,0,0],[9E+09,9E+09,9E+09,9E+09,9E+09,9E+09]],printSpeed,z0,bendedTool\WObj:=wobjpro1;
MoveL [[846,624.675,569.01],[0,0.997564,0.069756,0],[0,-1,0,0],[9E+09,9E+09,9E+09,9E+09,9E+09,9E+09]],printSpeed,z0,bendedTool\WObj:=wobjpro1;
MoveL [[846,575.325,569.01],[0,0.997564,0.069756,0],[0,-1,0,0],[9E+09,9E+09,9E+09,9E+09,9E+09,9E+09]],printSpeed,z0,bendedTool\WObj:=wobjpro1;
MoveL [[848,575.082,569.01],[0,0.997564,0.069756,0],[0,-1,0,0],[9E+09,9E+09,9E+09,9E+09,9E+09,9E+09]],printSpeed,z0,bendedTool\WObj:=wobjpro1;
MoveL [[848,624.918,569.01],[0,0.997564,0.069756,0],[0,-1,0,0],[9E+09,9E+09,9E+09,9E+09,9E+09,9E+09]],printSpeed,z0,bendedTool\WObj:=wobjpro1;
MoveL [[850,624.997,569.01],[0,0.997564,0.069756,0],[0,-1,0,0],[9E+09,9E+09,9E+09,9E+09,9E+09,9E+09]],printSpeed,z0,bendedTool\WObj:=wobjpro1;
MoveL [[850,575.003,569.01],[0,0.997564,0.069756,0],[0,-1,0,0],[9E+09,9E+09,9E+09,9E+09,9E+09,9E+09]],printSpeed,z0,bendedTool\WObj:=wobjpro1;
MoveL [[852,575.084,569.01],[0,0.997564,0.069756,0],[0,-1,0,0],[9E+09,9E+09,9E+09,9E+09,9E+09,9E+09]],printSpeed,z0,bendedTool\WObj:=wobjpro1;
MoveL [[852,624.916,569.01],[0,0.997564,0.069756,0],[0,-1,0,0],[9E+09,9E+09,9E+09,9E+09,9E+09,9E+09]],printSpeed,z0,bendedTool\WObj:=wobjpro1;
MoveL [[854,624.677,569.01],[0,0.997564,0.069756,0],[0,-1,0,0],[9E+09,9E+09,9E+09,9E+09,9E+09,9E+09]],printSpeed,z0,bendedTool\WObj:=wobjpro1;
MoveL [[854,575.323,569.01],[0,0.997564,0.069756,0],[0,-1,0,0],[9E+09,9E+09,9E+09,9E+09,9E+09,9E+09]],printSpeed,z0,bendedTool\WObj:=wobjpro1;
MoveL [[856,575.735,569.01],[0,0.997564,0.069756,0],[0,-1,0,0],[9E+09,9E+09,9E+09,9E+09,9E+09,9E+09]],printSpeed,z0,bendedTool\WObj:=wobjpro1;
MoveL [[856,624.265,569.01],[0,0.997564,0.069756,0],[0,-1,0,0],[9E+09,9E+09,9E+09,9E+09,9E+09,9E+09]],printSpeed,z0,bendedTool\WObj:=wobjpro1;
MoveL [[858,623.684,569.01],[0,0.997564,0.069756,0],[0,-1,0,0],[9E+09,9E+09,9E+09,9E+09,9E+09,9E+09]],printSpeed,z0,bendedTool\WObj:=wobjpro1;
MoveL [[858,576.316,569.01],[0,0.997564,0.069756,0],[0,-1,0,0],[9E+09,9E+09,9E+09,9E+09,9E+09,9E+09]],printSpeed,z0,bendedTool\WObj:=wobjpro1;
MoveL [[860,577.092,569.01],[0,0.997564,0.069756,0],[0,-1,0,0],[9E+09,9E+09,9E+09,9E+09,9E+09,9E+09]],printSpeed,z0,bendedTool\WObj:=wobjpro1;
MoveL [[860,622.908,569.01],[0,0.997564,0.069756,0],[0,-1,0,0],[9E+09,9E+09,9E+09,9E+09,9E+09,9E+09]],printSpeed,z0,bendedTool\WObj:=wobjpro1;
MoveL [[862,621.929,569.01],[0,0.997564,0.069756,0],[0,-1,0,0],[9E+09,9E+09,9E+09,9E+09,9E+09,9E+09]],printSpeed,z0,bendedTool\WObj:=wobjpro1;
MoveL [[862,578.071,569.01],[0,0.997564,0.069756,0],[0,-1,0,0],[9E+09,9E+09,9E+09,9E+09,9E+09,9E+09]],printSpeed,z0,bendedTool\WObj:=wobjpro1;
MoveL [[864,579.29,569.01],[0,0.997564,0.069756,0],[0,-1,0,0],[9E+09,9E+09,9E+09,9E+09,9E+09,9E+09]],printSpeed,z0,bendedTool\WObj:=wobjpro1;
MoveL [[864,620.71,569.01],[0,0.997564,0.069756,0],[0,-1,0,0],[9E+09,9E+09,9E+09,9E+09,9E+09,9E+09]],printSpeed,z0,bendedTool\WObj:=wobjpro1;
MoveL [[866,619.206,569.01],[0,0.997564,0.069756,0],[0,-1,0,0],[9E+09,9E+09,9E+09,9E+09,9E+09,9E+09]],printSpeed,z0,bendedTool\WObj:=wobjpro1;
MoveL [[866,580.794,569.01],[0,0.997564,0.069756,0],[0,-1,0,0],[9E+09,9E+09,9E+09,9E+09,9E+09,9E+09]],printSpeed,z0,bendedTool\WObj:=wobjpro1;
MoveL [[868,582.656,569.01],[0,0.997564,0.069756,0],[0,-1,0,0],[9E+09,9E+09,9E+09,9E+09,9E+09,9E+09]],printSpeed,z0,bendedTool\WObj:=wobjpro1;
MoveL [[868,617.344,569.01],[0,0.997564,0.069756,0],[0,-1,0,0],[9E+09,9E+09,9E+09,9E+09,9E+09,9E+09]],printSpeed,fine,bendedTool\WObj:=wobjpro1;
!stopContinuousWeld \delay:=delayOpenStop_0;
!MoveL [[868.000,617.344,669],[0.000000,0.997564,0.069756,0.000000],[0,-1,0,0],[9E9,9E9,9E9,9E9,9E9,9E9]],moveSpeed,z0,bendedTool,\WObj:=wobjpro1;
!MoveL [[870.000,614.994,669],[0.000000,0.997564,0.069756,0.000000],[0,-1,0,0],[9E9,9E9,9E9,9E9,9E9,9E9]],moveSpeed,z0,bendedTool,\WObj:=wobjpro1;
MoveL [[870,614.994,569.01],[0,0.997564,0.069756,0],[0,-1,0,0],[9E+09,9E+09,9E+09,9E+09,9E+09,9E+09]],moveSpeed,fine,bendedTool\WObj:=wobjpro1;
!startcontinuousweld; !layer  \delay:=delayOpenStart_0 \weldingProgram:=3 \weldId:="0000-0000-0005-0002";
!TPWrite "[55.0%] PRT0 LYR0 TRK5 (700.0mm)";
MoveL [[870,585.006,569.01],[0,0.997564,0.069756,0],[0,-1,0,0],[9E+09,9E+09,9E+09,9E+09,9E+09,9E+09]],printSpeed,fine,bendedTool\WObj:=wobjpro1;
!stopContinuousWeld \delay:=delayOpenStop_0;
!MoveL [[870.000,585.006,669],[0.000000,0.997564,0.069756,0.000000],[0,-1,0,0],[9E9,9E9,9E9,9E9,9E9,9E9]],moveSpeed,z0,bendedTool,\WObj:=wobjpro1;
!MoveL [[872.000,588.135,669],[0.000000,0.997564,0.069756,0.000000],[0,-1,0,0],[9E9,9E9,9E9,9E9,9E9,9E9]],moveSpeed,z0,bendedTool,\WObj:=wobjpro1;
MoveL [[872,588.135,569.01],[0,0.997564,0.069756,0],[0,-1,0,0],[9E+09,9E+09,9E+09,9E+09,9E+09,9E+09]],printSpeed,fine,bendedTool\WObj:=wobjpro1;
!startcontinuousweld; !layer  \delay:=delayOpenStart_0 \weldingProgram:=3 \weldId:="0000-0000-0006-0002";
TPWrite "[55.9%] PRT0 LYR0 TRK6 (700.0mm)";
MoveL [[872,611.865,569.01],[0,0.997564,0.069756,0],[0,-1,0,0],[9E+09,9E+09,9E+09,9E+09,9E+09,9E+09]],printSpeed,fine,bendedTool\WObj:=wobjpro1;
!stopContinuousWeld \delay:=delayOpenStop_0;
!MoveL [[872.000,611.865,669],[0.000000,0.997564,0.069756,0.000000],[0,-1,0,0],[9E9,9E9,9E9,9E9,9E9,9E9]],moveSpeed,z0,bendedTool,\WObj:=wobjpro1;
!MoveL [[874.000,606.981,669],[0.000000,0.997564,0.069756,0.000000],[0,-1,0,0],[9E9,9E9,9E9,9E9,9E9,9E9]],moveSpeed,z0,bendedTool,\WObj:=wobjpro1;
MoveL [[874,606.981,569.01],[0,0.997564,0.069756,0],[0,-1,0,0],[9E+09,9E+09,9E+09,9E+09,9E+09,9E+09]],printSpeed,fine,bendedTool\WObj:=wobjpro1;
!startcontinuousweld; !layer  \delay:=delayOpenStart_0 \weldingProgram:=3 \weldId:="0000-0000-0007-0002";
TPWrite "[56.8%] PRT0 LYR0 TRK7 (700.0mm)";
MoveL [[874,593.019,569.01],[0,0.997564,0.069756,0],[0,-1,0,0],[9E+09,9E+09,9E+09,9E+09,9E+09,9E+09]],printSpeed,fine,bendedTool\WObj:=wobjpro1;
stopContinuousWeld \delay:=delayOpenStop_0;
MoveL [[874,593.019,669],[0,0.997564,0.069756,0],[0,-1,0,0],[9E+09,9E+09,9E+09,9E+09,9E+09,9E+09]],moveSpeed,z0,bendedTool\WObj:=wobjpro1;
MoveL [[835.21,622.591,751.41],[0,0.997564,0.069756,0],[0,-1,0,0],[9E+09,9E+09,9E+09,9E+09,9E+09,9E+09]],moveSpeed,z0,bendedTool\WObj:=wobjpro1;

printSpeed := [12.0, 500.0, 10.0, 10.0];
tperase;
TPWrite "PRT0 is done printing";
tidyUp;
ENDPROC



PROC square()
VAR robtarget touchpoint:=[[850.000,575.000,565],[0.000000,0.997564,0.069756,0.000000],[0,-1,0,0],[9E9,9E9,9E9,9E9,9E9,9E9]];
interpassTemp := 200.0;
emissivity := 0.992;
MoveL [[861.996,625,700.01],[0,0.997564,0.069756,0],[0,-1,0,0],[9E+09,9E+09,9E+09,9E+09,9E+09,9E+09]],moveSpeed,z0,bendedTool\WObj:=wobjpro4;
serch_height 0,0,touchpoint,numtemp;
!(num ofx, num ofy, robtarget target, inout num zval)
wobjpro4.oframe.trans.z:=numtemp-569.010;



MoveL [[861.996,625,700.01],[0,0.997564,0.069756,0],[0,-1,0,0],[9E+09,9E+09,9E+09,9E+09,9E+09,9E+09]],moveSpeed,z0,bendedTool\WObj:=wobjpro4;
MoveL [[861.996,625,569.01],[0,0.997564,0.069756,0],[0,-1,0,0],[9E+09,9E+09,9E+09,9E+09,9E+09,9E+09]],moveSpeed,fine,bendedTool\WObj:=wobjpro4;
waitInterpass useTempSensor, wTime_25;
startcontinuousweld; !layer  \delay:=delayClosedStart_0 \weldId:="0000-0000-0000-0002";
TPWrite "[25.0%] PRT0 LYR0 TRK0 (569.0mm)";
MoveL [[875,625,569.01],[0,0.997564,0.069756,0],[0,-1,0,0],[9E+09,9E+09,9E+09,9E+09,9E+09,9E+09]],printSpeed,z0,bendedTool\WObj:=wobjpro4;
MoveL [[875,575,569.01],[0,0.997564,0.069756,0],[0,-1,0,0],[9E+09,9E+09,9E+09,9E+09,9E+09,9E+09]],printSpeed,z0,bendedTool\WObj:=wobjpro4;
MoveL [[825,575,569.01],[0,0.997564,0.069756,0],[0,-1,0,0],[9E+09,9E+09,9E+09,9E+09,9E+09,9E+09]],printSpeed,z0,bendedTool\WObj:=wobjpro4;
MoveL [[825,625,569.01],[0,0.997564,0.069756,0],[0,-1,0,0],[9E+09,9E+09,9E+09,9E+09,9E+09,9E+09]],printSpeed,z0,bendedTool\WObj:=wobjpro4;
MoveL [[861.996,625,569.01],[0,0.997564,0.069756,0],[0,-1,0,0],[9E+09,9E+09,9E+09,9E+09,9E+09,9E+09]],printSpeed,fine,bendedTool\WObj:=wobjpro4;
stopContinuousWeld \delay:=delayClosedStop_0;
TPERASE;
TPWrite "PRT0 is done printing";
MoveL [[861.996,625,669.01],[0,0.997564,0.069756,0],[0,-1,0,0],[9E+09,9E+09,9E+09,9E+09,9E+09,9E+09]],moveSpeed,z0,bendedTool\WObj:=wobjpro4;
tidyUp;
ENDPROC




PROC gaffel()
VAR robtarget touchpoint:=[[847.124,650.585,565],[0.000000,0.997564,0.069756,0.000000],[0,-1,0,0],[9E9,9E9,9E9,9E9,9E9,9E9]];
interpassTemp := 200.0;
emissivity := 0.992;
MoveL [[830.883,696.861,669.01],[0,0.997564,0.069756,0],[0,-1,0,0],[9E+09,9E+09,9E+09,9E+09,9E+09,9E+09]],moveSpeed,z0,bendedTool\WObj:=wobjpro2;
serch_height 0,0,touchpoint,numtemp;
!(num ofx, num ofy, robtarget target, inout num zval)
wobjpro2.oframe.trans.z:=numtemp-569.010;

MoveL [[830.883,696.861,669.01],[0,0.997564,0.069756,0],[0,-1,0,0],[9E+09,9E+09,9E+09,9E+09,9E+09,9E+09]],moveSpeed,z0,bendedTool\WObj:=wobjpro2;
MoveL [[830.883,696.861,569.01],[0,0.997564,0.069756,0],[0,-1,0,0],[9E+09,9E+09,9E+09,9E+09,9E+09,9E+09]],moveSpeed,fine,bendedTool\WObj:=wobjpro2;
waitInterpass useTempSensor, wTime_25;
startcontinuousweld; !layer  \delay:=delayOpenStart_0 \weldId:="0000-0000-0000-0002";
TPWrite "[2.5%] PRT0 LYR0 TRK0 (569.0mm)";
MoveL [[830.883,674.906,569.01],[0,0.997564,0.069756,0],[0,-1,0,0],[9E+09,9E+09,9E+09,9E+09,9E+09,9E+09]],printSpeed,z0,bendedTool\WObj:=wobjpro2;
MoveL [[830.918,674.068,569.01],[0,0.997564,0.069756,0],[0,-1,0,0],[9E+09,9E+09,9E+09,9E+09,9E+09,9E+09]],printSpeed,z0,bendedTool\WObj:=wobjpro2;
MoveL [[831.024,673.227,569.01],[0,0.997564,0.069756,0],[0,-1,0,0],[9E+09,9E+09,9E+09,9E+09,9E+09,9E+09]],printSpeed,z0,bendedTool\WObj:=wobjpro2;
MoveL [[831.2,672.407,569.01],[0,0.997564,0.069756,0],[0,-1,0,0],[9E+09,9E+09,9E+09,9E+09,9E+09,9E+09]],printSpeed,z0,bendedTool\WObj:=wobjpro2;
MoveL [[831.445,671.6,569.01],[0,0.997564,0.069756,0],[0,-1,0,0],[9E+09,9E+09,9E+09,9E+09,9E+09,9E+09]],printSpeed,z0,bendedTool\WObj:=wobjpro2;
MoveL [[831.757,670.817,569.01],[0,0.997564,0.069756,0],[0,-1,0,0],[9E+09,9E+09,9E+09,9E+09,9E+09,9E+09]],printSpeed,z0,bendedTool\WObj:=wobjpro2;
MoveL [[832.134,670.063,569.01],[0,0.997564,0.069756,0],[0,-1,0,0],[9E+09,9E+09,9E+09,9E+09,9E+09,9E+09]],printSpeed,z0,bendedTool\WObj:=wobjpro2;
MoveL [[832.573,669.343,569.01],[0,0.997564,0.069756,0],[0,-1,0,0],[9E+09,9E+09,9E+09,9E+09,9E+09,9E+09]],printSpeed,z0,bendedTool\WObj:=wobjpro2;
MoveL [[833.074,668.659,569.01],[0,0.997564,0.069756,0],[0,-1,0,0],[9E+09,9E+09,9E+09,9E+09,9E+09,9E+09]],printSpeed,z0,bendedTool\WObj:=wobjpro2;
MoveL [[845.809,652.739,569.01],[0,0.997564,0.069756,0],[0,-1,0,0],[9E+09,9E+09,9E+09,9E+09,9E+09,9E+09]],printSpeed,z0,bendedTool\WObj:=wobjpro2;
MoveL [[846.305,652.062,569.01],[0,0.997564,0.069756,0],[0,-1,0,0],[9E+09,9E+09,9E+09,9E+09,9E+09,9E+09]],printSpeed,z0,bendedTool\WObj:=wobjpro2;
MoveL [[846.745,651.343,569.01],[0,0.997564,0.069756,0],[0,-1,0,0],[9E+09,9E+09,9E+09,9E+09,9E+09,9E+09]],printSpeed,z0,bendedTool\WObj:=wobjpro2;
MoveL [[847.124,650.585,569.01],[0,0.997564,0.069756,0],[0,-1,0,0],[9E+09,9E+09,9E+09,9E+09,9E+09,9E+09]],printSpeed,z0,bendedTool\WObj:=wobjpro2;
MoveL [[847.435,649.806,569.01],[0,0.997564,0.069756,0],[0,-1,0,0],[9E+09,9E+09,9E+09,9E+09,9E+09,9E+09]],printSpeed,z0,bendedTool\WObj:=wobjpro2;
MoveL [[847.68,649,569.01],[0,0.997564,0.069756,0],[0,-1,0,0],[9E+09,9E+09,9E+09,9E+09,9E+09,9E+09]],printSpeed,z0,bendedTool\WObj:=wobjpro2;
MoveL [[847.857,648.175,569.01],[0,0.997564,0.069756,0],[0,-1,0,0],[9E+09,9E+09,9E+09,9E+09,9E+09,9E+09]],printSpeed,z0,bendedTool\WObj:=wobjpro2;
MoveL [[847.964,647.339,569.01],[0,0.997564,0.069756,0],[0,-1,0,0],[9E+09,9E+09,9E+09,9E+09,9E+09,9E+09]],printSpeed,z0,bendedTool\WObj:=wobjpro2;
MoveL [[848,646.497,569.01],[0,0.997564,0.069756,0],[0,-1,0,0],[9E+09,9E+09,9E+09,9E+09,9E+09,9E+09]],printSpeed,z0,bendedTool\WObj:=wobjpro2;
MoveL [[848,553.508,569.01],[0,0.997564,0.069756,0],[0,-1,0,0],[9E+09,9E+09,9E+09,9E+09,9E+09,9E+09]],printSpeed,z0,bendedTool\WObj:=wobjpro2;
MoveL [[847.965,552.669,569.01],[0,0.997564,0.069756,0],[0,-1,0,0],[9E+09,9E+09,9E+09,9E+09,9E+09,9E+09]],printSpeed,z0,bendedTool\WObj:=wobjpro2;
MoveL [[847.859,551.833,569.01],[0,0.997564,0.069756,0],[0,-1,0,0],[9E+09,9E+09,9E+09,9E+09,9E+09,9E+09]],printSpeed,z0,bendedTool\WObj:=wobjpro2;
MoveL [[847.683,551.009,569.01],[0,0.997564,0.069756,0],[0,-1,0,0],[9E+09,9E+09,9E+09,9E+09,9E+09,9E+09]],printSpeed,z0,bendedTool\WObj:=wobjpro2;
MoveL [[847.436,550.198,569.01],[0,0.997564,0.069756,0],[0,-1,0,0],[9E+09,9E+09,9E+09,9E+09,9E+09,9E+09]],printSpeed,z0,bendedTool\WObj:=wobjpro2;
MoveL [[847.126,549.418,569.01],[0,0.997564,0.069756,0],[0,-1,0,0],[9E+09,9E+09,9E+09,9E+09,9E+09,9E+09]],printSpeed,z0,bendedTool\WObj:=wobjpro2;
MoveL [[846.749,548.664,569.01],[0,0.997564,0.069756,0],[0,-1,0,0],[9E+09,9E+09,9E+09,9E+09,9E+09,9E+09]],printSpeed,z0,bendedTool\WObj:=wobjpro2;
MoveL [[846.307,547.941,569.01],[0,0.997564,0.069756,0],[0,-1,0,0],[9E+09,9E+09,9E+09,9E+09,9E+09,9E+09]],printSpeed,z0,bendedTool\WObj:=wobjpro2;
MoveL [[845.811,547.264,569.01],[0,0.997564,0.069756,0],[0,-1,0,0],[9E+09,9E+09,9E+09,9E+09,9E+09,9E+09]],printSpeed,z0,bendedTool\WObj:=wobjpro2;
MoveL [[833.074,531.341,569.01],[0,0.997564,0.069756,0],[0,-1,0,0],[9E+09,9E+09,9E+09,9E+09,9E+09,9E+09]],printSpeed,z0,bendedTool\WObj:=wobjpro2;
MoveL [[832.578,530.664,569.01],[0,0.997564,0.069756,0],[0,-1,0,0],[9E+09,9E+09,9E+09,9E+09,9E+09,9E+09]],printSpeed,z0,bendedTool\WObj:=wobjpro2;
MoveL [[832.136,529.941,569.01],[0,0.997564,0.069756,0],[0,-1,0,0],[9E+09,9E+09,9E+09,9E+09,9E+09,9E+09]],printSpeed,z0,bendedTool\WObj:=wobjpro2;
MoveL [[831.76,529.191,569.01],[0,0.997564,0.069756,0],[0,-1,0,0],[9E+09,9E+09,9E+09,9E+09,9E+09,9E+09]],printSpeed,z0,bendedTool\WObj:=wobjpro2;
MoveL [[831.448,528.408,569.01],[0,0.997564,0.069756,0],[0,-1,0,0],[9E+09,9E+09,9E+09,9E+09,9E+09,9E+09]],printSpeed,z0,bendedTool\WObj:=wobjpro2;
MoveL [[831.201,527.597,569.01],[0,0.997564,0.069756,0],[0,-1,0,0],[9E+09,9E+09,9E+09,9E+09,9E+09,9E+09]],printSpeed,z0,bendedTool\WObj:=wobjpro2;
MoveL [[831.025,526.777,569.01],[0,0.997564,0.069756,0],[0,-1,0,0],[9E+09,9E+09,9E+09,9E+09,9E+09,9E+09]],printSpeed,z0,bendedTool\WObj:=wobjpro2;
MoveL [[830.919,525.941,569.01],[0,0.997564,0.069756,0],[0,-1,0,0],[9E+09,9E+09,9E+09,9E+09,9E+09,9E+09]],printSpeed,z0,bendedTool\WObj:=wobjpro2;
MoveL [[830.883,525.098,569.01],[0,0.997564,0.069756,0],[0,-1,0,0],[9E+09,9E+09,9E+09,9E+09,9E+09,9E+09]],printSpeed,z0,bendedTool\WObj:=wobjpro2;
MoveL [[830.883,503.139,569.01],[0,0.997564,0.069756,0],[0,-1,0,0],[9E+09,9E+09,9E+09,9E+09,9E+09,9E+09]],printSpeed,fine,bendedTool\WObj:=wobjpro2;
stopContinuousWeld \delay:=delayOpenStop_0;
MoveL [[830.883,503.139,669.01],[0,0.997564,0.069756,0],[0,-1,0,0],[9E+09,9E+09,9E+09,9E+09,9E+09,9E+09]],moveSpeed,z0,bendedTool\WObj:=wobjpro2;
MoveL [[869.117,503.139,669.01],[0,0.997564,0.069756,0],[0,-1,0,0],[9E+09,9E+09,9E+09,9E+09,9E+09,9E+09]],moveSpeed,z0,bendedTool\WObj:=wobjpro2;
MoveL [[869.117,503.139,569.01],[0,0.997564,0.069756,0],[0,-1,0,0],[9E+09,9E+09,9E+09,9E+09,9E+09,9E+09]],moveSpeed,fine,bendedTool\WObj:=wobjpro2;
waitInterpass useTempSensor, wTime_25;
startcontinuousweld; !layer  \delay:=delayOpenStart_0 \weldId:="0000-0000-0001-0002";
TPWrite "[52.5%] PRT0 LYR0 TRK1 (569.0mm)";
MoveL [[869.117,525.094,569.01],[0,0.997564,0.069756,0],[0,-1,0,0],[9E+09,9E+09,9E+09,9E+09,9E+09,9E+09]],printSpeed,z0,bendedTool\WObj:=wobjpro2;
MoveL [[869.082,525.932,569.01],[0,0.997564,0.069756,0],[0,-1,0,0],[9E+09,9E+09,9E+09,9E+09,9E+09,9E+09]],printSpeed,z0,bendedTool\WObj:=wobjpro2;
MoveL [[868.976,526.769,569.01],[0,0.997564,0.069756,0],[0,-1,0,0],[9E+09,9E+09,9E+09,9E+09,9E+09,9E+09]],printSpeed,z0,bendedTool\WObj:=wobjpro2;
MoveL [[868.8,527.593,569.01],[0,0.997564,0.069756,0],[0,-1,0,0],[9E+09,9E+09,9E+09,9E+09,9E+09,9E+09]],printSpeed,z0,bendedTool\WObj:=wobjpro2;
MoveL [[868.555,528.4,569.01],[0,0.997564,0.069756,0],[0,-1,0,0],[9E+09,9E+09,9E+09,9E+09,9E+09,9E+09]],printSpeed,z0,bendedTool\WObj:=wobjpro2;
MoveL [[868.243,529.183,569.01],[0,0.997564,0.069756,0],[0,-1,0,0],[9E+09,9E+09,9E+09,9E+09,9E+09,9E+09]],printSpeed,z0,bendedTool\WObj:=wobjpro2;
MoveL [[867.866,529.937,569.01],[0,0.997564,0.069756,0],[0,-1,0,0],[9E+09,9E+09,9E+09,9E+09,9E+09,9E+09]],printSpeed,z0,bendedTool\WObj:=wobjpro2;
MoveL [[867.427,530.657,569.01],[0,0.997564,0.069756,0],[0,-1,0,0],[9E+09,9E+09,9E+09,9E+09,9E+09,9E+09]],printSpeed,z0,bendedTool\WObj:=wobjpro2;
MoveL [[866.929,531.337,569.01],[0,0.997564,0.069756,0],[0,-1,0,0],[9E+09,9E+09,9E+09,9E+09,9E+09,9E+09]],printSpeed,z0,bendedTool\WObj:=wobjpro2;
MoveL [[854.191,547.261,569.01],[0,0.997564,0.069756,0],[0,-1,0,0],[9E+09,9E+09,9E+09,9E+09,9E+09,9E+09]],printSpeed,z0,bendedTool\WObj:=wobjpro2;
MoveL [[853.695,547.938,569.01],[0,0.997564,0.069756,0],[0,-1,0,0],[9E+09,9E+09,9E+09,9E+09,9E+09,9E+09]],printSpeed,z0,bendedTool\WObj:=wobjpro2;
MoveL [[853.255,548.657,569.01],[0,0.997564,0.069756,0],[0,-1,0,0],[9E+09,9E+09,9E+09,9E+09,9E+09,9E+09]],printSpeed,z0,bendedTool\WObj:=wobjpro2;
MoveL [[852.878,549.411,569.01],[0,0.997564,0.069756,0],[0,-1,0,0],[9E+09,9E+09,9E+09,9E+09,9E+09,9E+09]],printSpeed,z0,bendedTool\WObj:=wobjpro2;
MoveL [[852.565,550.194,569.01],[0,0.997564,0.069756,0],[0,-1,0,0],[9E+09,9E+09,9E+09,9E+09,9E+09,9E+09]],printSpeed,z0,bendedTool\WObj:=wobjpro2;
MoveL [[852.318,551.004,569.01],[0,0.997564,0.069756,0],[0,-1,0,0],[9E+09,9E+09,9E+09,9E+09,9E+09,9E+09]],printSpeed,z0,bendedTool\WObj:=wobjpro2;
MoveL [[852.143,551.825,569.01],[0,0.997564,0.069756,0],[0,-1,0,0],[9E+09,9E+09,9E+09,9E+09,9E+09,9E+09]],printSpeed,z0,bendedTool\WObj:=wobjpro2;
MoveL [[852.036,552.661,569.01],[0,0.997564,0.069756,0],[0,-1,0,0],[9E+09,9E+09,9E+09,9E+09,9E+09,9E+09]],printSpeed,z0,bendedTool\WObj:=wobjpro2;
MoveL [[852,553.503,569.01],[0,0.997564,0.069756,0],[0,-1,0,0],[9E+09,9E+09,9E+09,9E+09,9E+09,9E+09]],printSpeed,z0,bendedTool\WObj:=wobjpro2;
MoveL [[852,646.492,569.01],[0,0.997564,0.069756,0],[0,-1,0,0],[9E+09,9E+09,9E+09,9E+09,9E+09,9E+09]],printSpeed,z0,bendedTool\WObj:=wobjpro2;
MoveL [[852.036,647.335,569.01],[0,0.997564,0.069756,0],[0,-1,0,0],[9E+09,9E+09,9E+09,9E+09,9E+09,9E+09]],printSpeed,z0,bendedTool\WObj:=wobjpro2;
MoveL [[852.142,648.171,569.01],[0,0.997564,0.069756,0],[0,-1,0,0],[9E+09,9E+09,9E+09,9E+09,9E+09,9E+09]],printSpeed,z0,bendedTool\WObj:=wobjpro2;
MoveL [[852.317,648.991,569.01],[0,0.997564,0.069756,0],[0,-1,0,0],[9E+09,9E+09,9E+09,9E+09,9E+09,9E+09]],printSpeed,z0,bendedTool\WObj:=wobjpro2;
MoveL [[852.562,649.798,569.01],[0,0.997564,0.069756,0],[0,-1,0,0],[9E+09,9E+09,9E+09,9E+09,9E+09,9E+09]],printSpeed,z0,bendedTool\WObj:=wobjpro2;
MoveL [[852.874,650.582,569.01],[0,0.997564,0.069756,0],[0,-1,0,0],[9E+09,9E+09,9E+09,9E+09,9E+09,9E+09]],printSpeed,z0,bendedTool\WObj:=wobjpro2;
MoveL [[853.253,651.339,569.01],[0,0.997564,0.069756,0],[0,-1,0,0],[9E+09,9E+09,9E+09,9E+09,9E+09,9E+09]],printSpeed,z0,bendedTool\WObj:=wobjpro2;
MoveL [[853.69,652.055,569.01],[0,0.997564,0.069756,0],[0,-1,0,0],[9E+09,9E+09,9E+09,9E+09,9E+09,9E+09]],printSpeed,z0,bendedTool\WObj:=wobjpro2;
MoveL [[854.191,652.739,569.01],[0,0.997564,0.069756,0],[0,-1,0,0],[9E+09,9E+09,9E+09,9E+09,9E+09,9E+09]],printSpeed,z0,bendedTool\WObj:=wobjpro2;
MoveL [[866.926,668.659,569.01],[0,0.997564,0.069756,0],[0,-1,0,0],[9E+09,9E+09,9E+09,9E+09,9E+09,9E+09]],printSpeed,z0,bendedTool\WObj:=wobjpro2;
MoveL [[867.425,669.339,569.01],[0,0.997564,0.069756,0],[0,-1,0,0],[9E+09,9E+09,9E+09,9E+09,9E+09,9E+09]],printSpeed,z0,bendedTool\WObj:=wobjpro2;
MoveL [[867.862,670.055,569.01],[0,0.997564,0.069756,0],[0,-1,0,0],[9E+09,9E+09,9E+09,9E+09,9E+09,9E+09]],printSpeed,z0,bendedTool\WObj:=wobjpro2;
MoveL [[868.241,670.813,569.01],[0,0.997564,0.069756,0],[0,-1,0,0],[9E+09,9E+09,9E+09,9E+09,9E+09,9E+09]],printSpeed,z0,bendedTool\WObj:=wobjpro2;
MoveL [[868.552,671.592,569.01],[0,0.997564,0.069756,0],[0,-1,0,0],[9E+09,9E+09,9E+09,9E+09,9E+09,9E+09]],printSpeed,z0,bendedTool\WObj:=wobjpro2;
MoveL [[868.798,672.399,569.01],[0,0.997564,0.069756,0],[0,-1,0,0],[9E+09,9E+09,9E+09,9E+09,9E+09,9E+09]],printSpeed,z0,bendedTool\WObj:=wobjpro2;
MoveL [[868.975,673.223,569.01],[0,0.997564,0.069756,0],[0,-1,0,0],[9E+09,9E+09,9E+09,9E+09,9E+09,9E+09]],printSpeed,z0,bendedTool\WObj:=wobjpro2;
MoveL [[869.082,674.063,569.01],[0,0.997564,0.069756,0],[0,-1,0,0],[9E+09,9E+09,9E+09,9E+09,9E+09,9E+09]],printSpeed,z0,bendedTool\WObj:=wobjpro2;
MoveL [[869.117,674.902,569.01],[0,0.997564,0.069756,0],[0,-1,0,0],[9E+09,9E+09,9E+09,9E+09,9E+09,9E+09]],printSpeed,z0,bendedTool\WObj:=wobjpro2;
MoveL [[869.117,696.861,569.01],[0,0.997564,0.069756,0],[0,-1,0,0],[9E+09,9E+09,9E+09,9E+09,9E+09,9E+09]],printSpeed,fine,bendedTool\WObj:=wobjpro2;
stopContinuousWeld \delay:=delayOpenStop_0;
TPerase;
TPWrite "PRT0 is done printing";
MoveL [[869.117,696.861,669.01],[0,0.997564,0.069756,0],[0,-1,0,0],[9E+09,9E+09,9E+09,9E+09,9E+09,9E+09]],moveSpeed,z0,bendedTool\WObj:=wobjpro2;
tidyUp;
ENDPROC









PROC dia100()
VAR robtarget touchpoint:=[[822.612,233.523,565],[0.000000,0.997564,0.069756,0.000000],[0,-1,0,0],[9E9,9E9,9E9,9E9,9E9,9E9]];
interpassTemp := 200.0;
emissivity := 0.992;
MoveL [[801.58,262.86,591.76],[0.000000652,0.997566,0.0697341,-0.000010747],[0,-1,0,0],[9E+09,9E+09,9E+09,9E+09,9E+09,9E+09]],moveSpeed,z0,bendedTool\WObj:=wobjpro3;
serch_height 0,0,touchpoint,numtemp;
!(num ofx, num ofy, robtarget target, inout num zval)
wobjpro3.oframe.trans.z:=numtemp-569.010;


MoveL [[801.58,262.86,591.76],[0.000000652,0.997566,0.0697341,-0.000010747],[0,-1,0,0],[9E+09,9E+09,9E+09,9E+09,9E+09,9E+09]],moveSpeed,z0,bendedTool\WObj:=wobjpro3;
MoveL [[801.575,262.89,569.01],[0,0.997564,0.069756,0],[0,-1,0,0],[9E+09,9E+09,9E+09,9E+09,9E+09,9E+09]],moveSpeed,fine,bendedTool\WObj:=wobjpro3;
waitInterpass useTempSensor, wTime_25;
startcontinuousweld; !layer  \delay:=delayClosedStart_0 \weldId:="0000-0000-0000-0002";
TPWrite "[1.0%] PRT0 LYR0 TRK0 (569.0mm)";
MoveL [[802.021,261.271,569.01],[0,0.997564,0.069756,0],[0,-1,0,0],[9E+09,9E+09,9E+09,9E+09,9E+09,9E+09]],printSpeed,z0,bendedTool\WObj:=wobjpro3;
MoveL [[802.522,259.667,569.01],[0,0.997564,0.069756,0],[0,-1,0,0],[9E+09,9E+09,9E+09,9E+09,9E+09,9E+09]],printSpeed,z0,bendedTool\WObj:=wobjpro3;
MoveL [[803.076,258.081,569.01],[0,0.997564,0.069756,0],[0,-1,0,0],[9E+09,9E+09,9E+09,9E+09,9E+09,9E+09]],printSpeed,z0,bendedTool\WObj:=wobjpro3;
MoveL [[803.682,256.515,569.01],[0,0.997564,0.069756,0],[0,-1,0,0],[9E+09,9E+09,9E+09,9E+09,9E+09,9E+09]],printSpeed,z0,bendedTool\WObj:=wobjpro3;
MoveL [[804.342,254.969,569.01],[0,0.997564,0.069756,0],[0,-1,0,0],[9E+09,9E+09,9E+09,9E+09,9E+09,9E+09]],printSpeed,z0,bendedTool\WObj:=wobjpro3;
MoveL [[805.052,253.447,569.01],[0,0.997564,0.069756,0],[0,-1,0,0],[9E+09,9E+09,9E+09,9E+09,9E+09,9E+09]],printSpeed,z0,bendedTool\WObj:=wobjpro3;
MoveL [[805.814,251.95,569.01],[0,0.997564,0.069756,0],[0,-1,0,0],[9E+09,9E+09,9E+09,9E+09,9E+09,9E+09]],printSpeed,z0,bendedTool\WObj:=wobjpro3;
MoveL [[806.625,250.479,569.01],[0,0.997564,0.069756,0],[0,-1,0,0],[9E+09,9E+09,9E+09,9E+09,9E+09,9E+09]],printSpeed,z0,bendedTool\WObj:=wobjpro3;
MoveL [[808.393,247.622,569.01],[0,0.997564,0.069756,0],[0,-1,0,0],[9E+09,9E+09,9E+09,9E+09,9E+09,9E+09]],printSpeed,z0,bendedTool\WObj:=wobjpro3;
MoveL [[807.485,249.036,569.01],[0,0.997564,0.069756,0],[0,-1,0,0],[9E+09,9E+09,9E+09,9E+09,9E+09,9E+09]],printSpeed,z0,bendedTool\WObj:=wobjpro3;
MoveL [[809.349,246.241,569.01],[0,0.997564,0.069756,0],[0,-1,0,0],[9E+09,9E+09,9E+09,9E+09,9E+09,9E+09]],printSpeed,z0,bendedTool\WObj:=wobjpro3;
MoveL [[810.35,244.891,569.01],[0,0.997564,0.069756,0],[0,-1,0,0],[9E+09,9E+09,9E+09,9E+09,9E+09,9E+09]],printSpeed,z0,bendedTool\WObj:=wobjpro3;
MoveL [[811.395,243.577,569.01],[0,0.997564,0.069756,0],[0,-1,0,0],[9E+09,9E+09,9E+09,9E+09,9E+09,9E+09]],printSpeed,z0,bendedTool\WObj:=wobjpro3;
MoveL [[812.485,242.298,569.01],[0,0.997564,0.069756,0],[0,-1,0,0],[9E+09,9E+09,9E+09,9E+09,9E+09,9E+09]],printSpeed,z0,bendedTool\WObj:=wobjpro3;
MoveL [[813.617,241.057,569.01],[0,0.997564,0.069756,0],[0,-1,0,0],[9E+09,9E+09,9E+09,9E+09,9E+09,9E+09]],printSpeed,z0,bendedTool\WObj:=wobjpro3;
MoveL [[814.789,239.854,569.01],[0,0.997564,0.069756,0],[0,-1,0,0],[9E+09,9E+09,9E+09,9E+09,9E+09,9E+09]],printSpeed,z0,bendedTool\WObj:=wobjpro3;
MoveL [[816.002,238.691,569.01],[0,0.997564,0.069756,0],[0,-1,0,0],[9E+09,9E+09,9E+09,9E+09,9E+09,9E+09]],printSpeed,z0,bendedTool\WObj:=wobjpro3;
MoveL [[817.253,237.57,569.01],[0,0.997564,0.069756,0],[0,-1,0,0],[9E+09,9E+09,9E+09,9E+09,9E+09,9E+09]],printSpeed,z0,bendedTool\WObj:=wobjpro3;
MoveL [[818.541,236.491,569.01],[0,0.997564,0.069756,0],[0,-1,0,0],[9E+09,9E+09,9E+09,9E+09,9E+09,9E+09]],printSpeed,z0,bendedTool\WObj:=wobjpro3;
MoveL [[819.864,235.456,569.01],[0,0.997564,0.069756,0],[0,-1,0,0],[9E+09,9E+09,9E+09,9E+09,9E+09,9E+09]],printSpeed,z0,bendedTool\WObj:=wobjpro3;
MoveL [[821.222,234.467,569.01],[0,0.997564,0.069756,0],[0,-1,0,0],[9E+09,9E+09,9E+09,9E+09,9E+09,9E+09]],printSpeed,z0,bendedTool\WObj:=wobjpro3;
MoveL [[822.612,233.523,569.01],[0,0.997564,0.069756,0],[0,-1,0,0],[9E+09,9E+09,9E+09,9E+09,9E+09,9E+09]],printSpeed,z0,bendedTool\WObj:=wobjpro3;
MoveL [[824.032,232.627,569.01],[0,0.997564,0.069756,0],[0,-1,0,0],[9E+09,9E+09,9E+09,9E+09,9E+09,9E+09]],printSpeed,z0,bendedTool\WObj:=wobjpro3;
MoveL [[825.483,231.779,569.01],[0,0.997564,0.069756,0],[0,-1,0,0],[9E+09,9E+09,9E+09,9E+09,9E+09,9E+09]],printSpeed,z0,bendedTool\WObj:=wobjpro3;
MoveL [[826.96,230.98,569.01],[0,0.997564,0.069756,0],[0,-1,0,0],[9E+09,9E+09,9E+09,9E+09,9E+09,9E+09]],printSpeed,z0,bendedTool\WObj:=wobjpro3;
MoveL [[828.464,230.231,569.01],[0,0.997564,0.069756,0],[0,-1,0,0],[9E+09,9E+09,9E+09,9E+09,9E+09,9E+09]],printSpeed,z0,bendedTool\WObj:=wobjpro3;
MoveL [[829.992,229.533,569.01],[0,0.997564,0.069756,0],[0,-1,0,0],[9E+09,9E+09,9E+09,9E+09,9E+09,9E+09]],printSpeed,z0,bendedTool\WObj:=wobjpro3;
MoveL [[831.543,228.887,569.01],[0,0.997564,0.069756,0],[0,-1,0,0],[9E+09,9E+09,9E+09,9E+09,9E+09,9E+09]],printSpeed,z0,bendedTool\WObj:=wobjpro3;
MoveL [[833.114,228.293,569.01],[0,0.997564,0.069756,0],[0,-1,0,0],[9E+09,9E+09,9E+09,9E+09,9E+09,9E+09]],printSpeed,z0,bendedTool\WObj:=wobjpro3;
MoveL [[834.705,227.753,569.01],[0,0.997564,0.069756,0],[0,-1,0,0],[9E+09,9E+09,9E+09,9E+09,9E+09,9E+09]],printSpeed,z0,bendedTool\WObj:=wobjpro3;
MoveL [[836.313,227.266,569.01],[0,0.997564,0.069756,0],[0,-1,0,0],[9E+09,9E+09,9E+09,9E+09,9E+09,9E+09]],printSpeed,z0,bendedTool\WObj:=wobjpro3;
MoveL [[837.944,226.832,569.01],[0,0.997564,0.069756,0],[0,-1,0,0],[9E+09,9E+09,9E+09,9E+09,9E+09,9E+09]],printSpeed,z0,bendedTool\WObj:=wobjpro3;
MoveL [[839.573,226.456,569.01],[0,0.997564,0.069756,0],[0,-1,0,0],[9E+09,9E+09,9E+09,9E+09,9E+09,9E+09]],printSpeed,z0,bendedTool\WObj:=wobjpro3;
MoveL [[841.222,226.133,569.01],[0,0.997564,0.069756,0],[0,-1,0,0],[9E+09,9E+09,9E+09,9E+09,9E+09,9E+09]],printSpeed,z0,bendedTool\WObj:=wobjpro3;
MoveL [[842.88,225.866,569.01],[0,0.997564,0.069756,0],[0,-1,0,0],[9E+09,9E+09,9E+09,9E+09,9E+09,9E+09]],printSpeed,z0,bendedTool\WObj:=wobjpro3;
MoveL [[844.547,225.655,569.01],[0,0.997564,0.069756,0],[0,-1,0,0],[9E+09,9E+09,9E+09,9E+09,9E+09,9E+09]],printSpeed,z0,bendedTool\WObj:=wobjpro3;
MoveL [[846.22,225.5,569.01],[0,0.997564,0.069756,0],[0,-1,0,0],[9E+09,9E+09,9E+09,9E+09,9E+09,9E+09]],printSpeed,z0,bendedTool\WObj:=wobjpro3;
MoveL [[847.897,225.401,569.01],[0,0.997564,0.069756,0],[0,-1,0,0],[9E+09,9E+09,9E+09,9E+09,9E+09,9E+09]],printSpeed,z0,bendedTool\WObj:=wobjpro3;
MoveL [[849.584,225.359,569.01],[0,0.997564,0.069756,0],[0,-1,0,0],[9E+09,9E+09,9E+09,9E+09,9E+09,9E+09]],printSpeed,z0,bendedTool\WObj:=wobjpro3;
MoveL [[851.256,225.373,569.01],[0,0.997564,0.069756,0],[0,-1,0,0],[9E+09,9E+09,9E+09,9E+09,9E+09,9E+09]],printSpeed,z0,bendedTool\WObj:=wobjpro3;
MoveL [[852.934,225.444,569.01],[0,0.997564,0.069756,0],[0,-1,0,0],[9E+09,9E+09,9E+09,9E+09,9E+09,9E+09]],printSpeed,z0,bendedTool\WObj:=wobjpro3;
MoveL [[854.609,225.571,569.01],[0,0.997564,0.069756,0],[0,-1,0,0],[9E+09,9E+09,9E+09,9E+09,9E+09,9E+09]],printSpeed,z0,bendedTool\WObj:=wobjpro3;
MoveL [[856.279,225.754,569.01],[0,0.997564,0.069756,0],[0,-1,0,0],[9E+09,9E+09,9E+09,9E+09,9E+09,9E+09]],printSpeed,z0,bendedTool\WObj:=wobjpro3;
MoveL [[857.942,225.993,569.01],[0,0.997564,0.069756,0],[0,-1,0,0],[9E+09,9E+09,9E+09,9E+09,9E+09,9E+09]],printSpeed,z0,bendedTool\WObj:=wobjpro3;
MoveL [[859.596,226.288,569.01],[0,0.997564,0.069756,0],[0,-1,0,0],[9E+09,9E+09,9E+09,9E+09,9E+09,9E+09]],printSpeed,z0,bendedTool\WObj:=wobjpro3;
MoveL [[861.239,226.638,569.01],[0,0.997564,0.069756,0],[0,-1,0,0],[9E+09,9E+09,9E+09,9E+09,9E+09,9E+09]],printSpeed,z0,bendedTool\WObj:=wobjpro3;
MoveL [[862.869,227.043,569.01],[0,0.997564,0.069756,0],[0,-1,0,0],[9E+09,9E+09,9E+09,9E+09,9E+09,9E+09]],printSpeed,z0,bendedTool\WObj:=wobjpro3;
MoveL [[864.485,227.503,569.01],[0,0.997564,0.069756,0],[0,-1,0,0],[9E+09,9E+09,9E+09,9E+09,9E+09,9E+09]],printSpeed,z0,bendedTool\WObj:=wobjpro3;
MoveL [[866.085,228.016,569.01],[0,0.997564,0.069756,0],[0,-1,0,0],[9E+09,9E+09,9E+09,9E+09,9E+09,9E+09]],printSpeed,z0,bendedTool\WObj:=wobjpro3;
MoveL [[867.666,228.584,569.01],[0,0.997564,0.069756,0],[0,-1,0,0],[9E+09,9E+09,9E+09,9E+09,9E+09,9E+09]],printSpeed,z0,bendedTool\WObj:=wobjpro3;
MoveL [[869.227,229.204,569.01],[0,0.997564,0.069756,0],[0,-1,0,0],[9E+09,9E+09,9E+09,9E+09,9E+09,9E+09]],printSpeed,z0,bendedTool\WObj:=wobjpro3;
MoveL [[870.774,229.879,569.01],[0,0.997564,0.069756,0],[0,-1,0,0],[9E+09,9E+09,9E+09,9E+09,9E+09,9E+09]],printSpeed,z0,bendedTool\WObj:=wobjpro3;
MoveL [[872.283,230.599,569.01],[0,0.997564,0.069756,0],[0,-1,0,0],[9E+09,9E+09,9E+09,9E+09,9E+09,9E+09]],printSpeed,z0,bendedTool\WObj:=wobjpro3;
MoveL [[873.774,231.373,569.01],[0,0.997564,0.069756,0],[0,-1,0,0],[9E+09,9E+09,9E+09,9E+09,9E+09,9E+09]],printSpeed,z0,bendedTool\WObj:=wobjpro3;
MoveL [[875.238,232.197,569.01],[0,0.997564,0.069756,0],[0,-1,0,0],[9E+09,9E+09,9E+09,9E+09,9E+09,9E+09]],printSpeed,z0,bendedTool\WObj:=wobjpro3;
MoveL [[876.674,233.069,569.01],[0,0.997564,0.069756,0],[0,-1,0,0],[9E+09,9E+09,9E+09,9E+09,9E+09,9E+09]],printSpeed,z0,bendedTool\WObj:=wobjpro3;
MoveL [[878.079,233.989,569.01],[0,0.997564,0.069756,0],[0,-1,0,0],[9E+09,9E+09,9E+09,9E+09,9E+09,9E+09]],printSpeed,z0,bendedTool\WObj:=wobjpro3;
MoveL [[879.453,234.956,569.01],[0,0.997564,0.069756,0],[0,-1,0,0],[9E+09,9E+09,9E+09,9E+09,9E+09,9E+09]],printSpeed,z0,bendedTool\WObj:=wobjpro3;
MoveL [[880.794,235.968,569.01],[0,0.997564,0.069756,0],[0,-1,0,0],[9E+09,9E+09,9E+09,9E+09,9E+09,9E+09]],printSpeed,z0,bendedTool\WObj:=wobjpro3;
MoveL [[882.1,237.025,569.01],[0,0.997564,0.069756,0],[0,-1,0,0],[9E+09,9E+09,9E+09,9E+09,9E+09,9E+09]],printSpeed,z0,bendedTool\WObj:=wobjpro3;
MoveL [[883.369,238.125,569.01],[0,0.997564,0.069756,0],[0,-1,0,0],[9E+09,9E+09,9E+09,9E+09,9E+09,9E+09]],printSpeed,z0,bendedTool\WObj:=wobjpro3;
MoveL [[884.601,239.267,569.01],[0,0.997564,0.069756,0],[0,-1,0,0],[9E+09,9E+09,9E+09,9E+09,9E+09,9E+09]],printSpeed,z0,bendedTool\WObj:=wobjpro3;
MoveL [[885.794,240.45,569.01],[0,0.997564,0.069756,0],[0,-1,0,0],[9E+09,9E+09,9E+09,9E+09,9E+09,9E+09]],printSpeed,z0,bendedTool\WObj:=wobjpro3;
MoveL [[886.946,241.673,569.01],[0,0.997564,0.069756,0],[0,-1,0,0],[9E+09,9E+09,9E+09,9E+09,9E+09,9E+09]],printSpeed,z0,bendedTool\WObj:=wobjpro3;
MoveL [[888.057,242.933,569.01],[0,0.997564,0.069756,0],[0,-1,0,0],[9E+09,9E+09,9E+09,9E+09,9E+09,9E+09]],printSpeed,z0,bendedTool\WObj:=wobjpro3;
MoveL [[889.125,244.23,569.01],[0,0.997564,0.069756,0],[0,-1,0,0],[9E+09,9E+09,9E+09,9E+09,9E+09,9E+09]],printSpeed,z0,bendedTool\WObj:=wobjpro3;
MoveL [[890.149,245.562,569.01],[0,0.997564,0.069756,0],[0,-1,0,0],[9E+09,9E+09,9E+09,9E+09,9E+09,9E+09]],printSpeed,z0,bendedTool\WObj:=wobjpro3;
MoveL [[891.127,246.927,569.01],[0,0.997564,0.069756,0],[0,-1,0,0],[9E+09,9E+09,9E+09,9E+09,9E+09,9E+09]],printSpeed,z0,bendedTool\WObj:=wobjpro3;
MoveL [[892.059,248.325,569.01],[0,0.997564,0.069756,0],[0,-1,0,0],[9E+09,9E+09,9E+09,9E+09,9E+09,9E+09]],printSpeed,z0,bendedTool\WObj:=wobjpro3;
MoveL [[892.943,249.754,569.01],[0,0.997564,0.069756,0],[0,-1,0,0],[9E+09,9E+09,9E+09,9E+09,9E+09,9E+09]],printSpeed,z0,bendedTool\WObj:=wobjpro3;
MoveL [[893.779,251.211,569.01],[0,0.997564,0.069756,0],[0,-1,0,0],[9E+09,9E+09,9E+09,9E+09,9E+09,9E+09]],printSpeed,z0,bendedTool\WObj:=wobjpro3;
MoveL [[893.783,251.218,569.01],[0,0.997564,0.069756,0],[0,-1,0,0],[9E+09,9E+09,9E+09,9E+09,9E+09,9E+09]],printSpeed,z0,bendedTool\WObj:=wobjpro3;
MoveL [[894.569,252.703,569.01],[0,0.997564,0.069756,0],[0,-1,0,0],[9E+09,9E+09,9E+09,9E+09,9E+09,9E+09]],printSpeed,z0,bendedTool\WObj:=wobjpro3;
MoveL [[895.305,254.213,569.01],[0,0.997564,0.069756,0],[0,-1,0,0],[9E+09,9E+09,9E+09,9E+09,9E+09,9E+09]],printSpeed,z0,bendedTool\WObj:=wobjpro3;
MoveL [[895.987,255.739,569.01],[0,0.997564,0.069756,0],[0,-1,0,0],[9E+09,9E+09,9E+09,9E+09,9E+09,9E+09]],printSpeed,z0,bendedTool\WObj:=wobjpro3;
MoveL [[896.623,257.303,569.01],[0,0.997564,0.069756,0],[0,-1,0,0],[9E+09,9E+09,9E+09,9E+09,9E+09,9E+09]],printSpeed,z0,bendedTool\WObj:=wobjpro3;
MoveL [[897.2,258.872,569.01],[0,0.997564,0.069756,0],[0,-1,0,0],[9E+09,9E+09,9E+09,9E+09,9E+09,9E+09]],printSpeed,z0,bendedTool\WObj:=wobjpro3;
MoveL [[897.727,260.467,569.01],[0,0.997564,0.069756,0],[0,-1,0,0],[9E+09,9E+09,9E+09,9E+09,9E+09,9E+09]],printSpeed,z0,bendedTool\WObj:=wobjpro3;
MoveL [[898.201,262.079,569.01],[0,0.997564,0.069756,0],[0,-1,0,0],[9E+09,9E+09,9E+09,9E+09,9E+09,9E+09]],printSpeed,z0,bendedTool\WObj:=wobjpro3;
MoveL [[898.621,263.714,569.01],[0,0.997564,0.069756,0],[0,-1,0,0],[9E+09,9E+09,9E+09,9E+09,9E+09,9E+09]],printSpeed,z0,bendedTool\WObj:=wobjpro3;
MoveL [[898.985,265.354,569.01],[0,0.997564,0.069756,0],[0,-1,0,0],[9E+09,9E+09,9E+09,9E+09,9E+09,9E+09]],printSpeed,z0,bendedTool\WObj:=wobjpro3;
MoveL [[899.292,266.997,569.01],[0,0.997564,0.069756,0],[0,-1,0,0],[9E+09,9E+09,9E+09,9E+09,9E+09,9E+09]],printSpeed,z0,bendedTool\WObj:=wobjpro3;
MoveL [[899.545,268.658,569.01],[0,0.997564,0.069756,0],[0,-1,0,0],[9E+09,9E+09,9E+09,9E+09,9E+09,9E+09]],printSpeed,z0,bendedTool\WObj:=wobjpro3;
MoveL [[899.742,270.326,569.01],[0,0.997564,0.069756,0],[0,-1,0,0],[9E+09,9E+09,9E+09,9E+09,9E+09,9E+09]],printSpeed,z0,bendedTool\WObj:=wobjpro3;
MoveL [[899.883,272,569.01],[0,0.997564,0.069756,0],[0,-1,0,0],[9E+09,9E+09,9E+09,9E+09,9E+09,9E+09]],printSpeed,z0,bendedTool\WObj:=wobjpro3;
MoveL [[899.968,273.678,569.01],[0,0.997564,0.069756,0],[0,-1,0,0],[9E+09,9E+09,9E+09,9E+09,9E+09,9E+09]],printSpeed,z0,bendedTool\WObj:=wobjpro3;
MoveL [[899.996,275.357,569.01],[0,0.997564,0.069756,0],[0,-1,0,0],[9E+09,9E+09,9E+09,9E+09,9E+09,9E+09]],printSpeed,z0,bendedTool\WObj:=wobjpro3;
MoveL [[899.968,277.037,569.01],[0,0.997564,0.069756,0],[0,-1,0,0],[9E+09,9E+09,9E+09,9E+09,9E+09,9E+09]],printSpeed,z0,bendedTool\WObj:=wobjpro3;
MoveL [[899.883,278.715,569.01],[0,0.997564,0.069756,0],[0,-1,0,0],[9E+09,9E+09,9E+09,9E+09,9E+09,9E+09]],printSpeed,z0,bendedTool\WObj:=wobjpro3;
MoveL [[899.742,280.389,569.01],[0,0.997564,0.069756,0],[0,-1,0,0],[9E+09,9E+09,9E+09,9E+09,9E+09,9E+09]],printSpeed,z0,bendedTool\WObj:=wobjpro3;
MoveL [[899.545,282.057,569.01],[0,0.997564,0.069756,0],[0,-1,0,0],[9E+09,9E+09,9E+09,9E+09,9E+09,9E+09]],printSpeed,z0,bendedTool\WObj:=wobjpro3;
MoveL [[899.292,283.718,569.01],[0,0.997564,0.069756,0],[0,-1,0,0],[9E+09,9E+09,9E+09,9E+09,9E+09,9E+09]],printSpeed,z0,bendedTool\WObj:=wobjpro3;
MoveL [[898.983,285.369,569.01],[0,0.997564,0.069756,0],[0,-1,0,0],[9E+09,9E+09,9E+09,9E+09,9E+09,9E+09]],printSpeed,z0,bendedTool\WObj:=wobjpro3;
MoveL [[898.619,287.009,569.01],[0,0.997564,0.069756,0],[0,-1,0,0],[9E+09,9E+09,9E+09,9E+09,9E+09,9E+09]],printSpeed,z0,bendedTool\WObj:=wobjpro3;
MoveL [[898.198,288.644,569.01],[0,0.997564,0.069756,0],[0,-1,0,0],[9E+09,9E+09,9E+09,9E+09,9E+09,9E+09]],printSpeed,z0,bendedTool\WObj:=wobjpro3;
MoveL [[897.727,290.248,569.01],[0,0.997564,0.069756,0],[0,-1,0,0],[9E+09,9E+09,9E+09,9E+09,9E+09,9E+09]],printSpeed,z0,bendedTool\WObj:=wobjpro3;
MoveL [[897.2,291.843,569.01],[0,0.997564,0.069756,0],[0,-1,0,0],[9E+09,9E+09,9E+09,9E+09,9E+09,9E+09]],printSpeed,z0,bendedTool\WObj:=wobjpro3;
MoveL [[896.62,293.419,569.01],[0,0.997564,0.069756,0],[0,-1,0,0],[9E+09,9E+09,9E+09,9E+09,9E+09,9E+09]],printSpeed,z0,bendedTool\WObj:=wobjpro3;
MoveL [[895.987,294.975,569.01],[0,0.997564,0.069756,0],[0,-1,0,0],[9E+09,9E+09,9E+09,9E+09,9E+09,9E+09]],printSpeed,z0,bendedTool\WObj:=wobjpro3;
MoveL [[895.302,296.509,569.01],[0,0.997564,0.069756,0],[0,-1,0,0],[9E+09,9E+09,9E+09,9E+09,9E+09,9E+09]],printSpeed,z0,bendedTool\WObj:=wobjpro3;
MoveL [[894.565,298.019,569.01],[0,0.997564,0.069756,0],[0,-1,0,0],[9E+09,9E+09,9E+09,9E+09,9E+09,9E+09]],printSpeed,z0,bendedTool\WObj:=wobjpro3;
MoveL [[893.779,299.504,569.01],[0,0.997564,0.069756,0],[0,-1,0,0],[9E+09,9E+09,9E+09,9E+09,9E+09,9E+09]],printSpeed,z0,bendedTool\WObj:=wobjpro3;
MoveL [[892.943,300.961,569.01],[0,0.997564,0.069756,0],[0,-1,0,0],[9E+09,9E+09,9E+09,9E+09,9E+09,9E+09]],printSpeed,z0,bendedTool\WObj:=wobjpro3;
MoveL [[892.059,302.389,569.01],[0,0.997564,0.069756,0],[0,-1,0,0],[9E+09,9E+09,9E+09,9E+09,9E+09,9E+09]],printSpeed,z0,bendedTool\WObj:=wobjpro3;
MoveL [[891.127,303.787,569.01],[0,0.997564,0.069756,0],[0,-1,0,0],[9E+09,9E+09,9E+09,9E+09,9E+09,9E+09]],printSpeed,z0,bendedTool\WObj:=wobjpro3;
MoveL [[890.149,305.153,569.01],[0,0.997564,0.069756,0],[0,-1,0,0],[9E+09,9E+09,9E+09,9E+09,9E+09,9E+09]],printSpeed,z0,bendedTool\WObj:=wobjpro3;
MoveL [[889.125,306.485,569.01],[0,0.997564,0.069756,0],[0,-1,0,0],[9E+09,9E+09,9E+09,9E+09,9E+09,9E+09]],printSpeed,z0,bendedTool\WObj:=wobjpro3;
MoveL [[888.057,307.782,569.01],[0,0.997564,0.069756,0],[0,-1,0,0],[9E+09,9E+09,9E+09,9E+09,9E+09,9E+09]],printSpeed,z0,bendedTool\WObj:=wobjpro3;
MoveL [[886.946,309.042,569.01],[0,0.997564,0.069756,0],[0,-1,0,0],[9E+09,9E+09,9E+09,9E+09,9E+09,9E+09]],printSpeed,z0,bendedTool\WObj:=wobjpro3;
MoveL [[885.794,310.264,569.01],[0,0.997564,0.069756,0],[0,-1,0,0],[9E+09,9E+09,9E+09,9E+09,9E+09,9E+09]],printSpeed,z0,bendedTool\WObj:=wobjpro3;
MoveL [[884.601,311.447,569.01],[0,0.997564,0.069756,0],[0,-1,0,0],[9E+09,9E+09,9E+09,9E+09,9E+09,9E+09]],printSpeed,z0,bendedTool\WObj:=wobjpro3;
MoveL [[883.369,312.589,569.01],[0,0.997564,0.069756,0],[0,-1,0,0],[9E+09,9E+09,9E+09,9E+09,9E+09,9E+09]],printSpeed,z0,bendedTool\WObj:=wobjpro3;
MoveL [[882.1,313.69,569.01],[0,0.997564,0.069756,0],[0,-1,0,0],[9E+09,9E+09,9E+09,9E+09,9E+09,9E+09]],printSpeed,z0,bendedTool\WObj:=wobjpro3;
MoveL [[880.787,314.751,569.01],[0,0.997564,0.069756,0],[0,-1,0,0],[9E+09,9E+09,9E+09,9E+09,9E+09,9E+09]],printSpeed,z0,bendedTool\WObj:=wobjpro3;
MoveL [[879.446,315.764,569.01],[0,0.997564,0.069756,0],[0,-1,0,0],[9E+09,9E+09,9E+09,9E+09,9E+09,9E+09]],printSpeed,z0,bendedTool\WObj:=wobjpro3;
MoveL [[878.079,316.726,569.01],[0,0.997564,0.069756,0],[0,-1,0,0],[9E+09,9E+09,9E+09,9E+09,9E+09,9E+09]],printSpeed,z0,bendedTool\WObj:=wobjpro3;
MoveL [[876.667,317.65,569.01],[0,0.997564,0.069756,0],[0,-1,0,0],[9E+09,9E+09,9E+09,9E+09,9E+09,9E+09]],printSpeed,z0,bendedTool\WObj:=wobjpro3;
MoveL [[875.238,318.518,569.01],[0,0.997564,0.069756,0],[0,-1,0,0],[9E+09,9E+09,9E+09,9E+09,9E+09,9E+09]],printSpeed,z0,bendedTool\WObj:=wobjpro3;
MoveL [[873.774,319.342,569.01],[0,0.997564,0.069756,0],[0,-1,0,0],[9E+09,9E+09,9E+09,9E+09,9E+09,9E+09]],printSpeed,z0,bendedTool\WObj:=wobjpro3;
MoveL [[872.283,320.115,569.01],[0,0.997564,0.069756,0],[0,-1,0,0],[9E+09,9E+09,9E+09,9E+09,9E+09,9E+09]],printSpeed,z0,bendedTool\WObj:=wobjpro3;
MoveL [[870.767,320.839,569.01],[0,0.997564,0.069756,0],[0,-1,0,0],[9E+09,9E+09,9E+09,9E+09,9E+09,9E+09]],printSpeed,z0,bendedTool\WObj:=wobjpro3;
MoveL [[869.227,321.511,569.01],[0,0.997564,0.069756,0],[0,-1,0,0],[9E+09,9E+09,9E+09,9E+09,9E+09,9E+09]],printSpeed,z0,bendedTool\WObj:=wobjpro3;
MoveL [[867.666,322.131,569.01],[0,0.997564,0.069756,0],[0,-1,0,0],[9E+09,9E+09,9E+09,9E+09,9E+09,9E+09]],printSpeed,z0,bendedTool\WObj:=wobjpro3;
MoveL [[866.085,322.698,569.01],[0,0.997564,0.069756,0],[0,-1,0,0],[9E+09,9E+09,9E+09,9E+09,9E+09,9E+09]],printSpeed,z0,bendedTool\WObj:=wobjpro3;
MoveL [[864.485,323.212,569.01],[0,0.997564,0.069756,0],[0,-1,0,0],[9E+09,9E+09,9E+09,9E+09,9E+09,9E+09]],printSpeed,z0,bendedTool\WObj:=wobjpro3;
MoveL [[862.869,323.672,569.01],[0,0.997564,0.069756,0],[0,-1,0,0],[9E+09,9E+09,9E+09,9E+09,9E+09,9E+09]],printSpeed,z0,bendedTool\WObj:=wobjpro3;
MoveL [[861.239,324.077,569.01],[0,0.997564,0.069756,0],[0,-1,0,0],[9E+09,9E+09,9E+09,9E+09,9E+09,9E+09]],printSpeed,z0,bendedTool\WObj:=wobjpro3;
MoveL [[859.596,324.427,569.01],[0,0.997564,0.069756,0],[0,-1,0,0],[9E+09,9E+09,9E+09,9E+09,9E+09,9E+09]],printSpeed,z0,bendedTool\WObj:=wobjpro3;
MoveL [[857.942,324.722,569.01],[0,0.997564,0.069756,0],[0,-1,0,0],[9E+09,9E+09,9E+09,9E+09,9E+09,9E+09]],printSpeed,z0,bendedTool\WObj:=wobjpro3;
MoveL [[856.279,324.961,569.01],[0,0.997564,0.069756,0],[0,-1,0,0],[9E+09,9E+09,9E+09,9E+09,9E+09,9E+09]],printSpeed,z0,bendedTool\WObj:=wobjpro3;
MoveL [[854.609,325.144,569.01],[0,0.997564,0.069756,0],[0,-1,0,0],[9E+09,9E+09,9E+09,9E+09,9E+09,9E+09]],printSpeed,z0,bendedTool\WObj:=wobjpro3;
MoveL [[852.926,325.271,569.01],[0,0.997564,0.069756,0],[0,-1,0,0],[9E+09,9E+09,9E+09,9E+09,9E+09,9E+09]],printSpeed,z0,bendedTool\WObj:=wobjpro3;
MoveL [[851.256,325.341,569.01],[0,0.997564,0.069756,0],[0,-1,0,0],[9E+09,9E+09,9E+09,9E+09,9E+09,9E+09]],printSpeed,z0,bendedTool\WObj:=wobjpro3;
MoveL [[849.576,325.356,569.01],[0,0.997564,0.069756,0],[0,-1,0,0],[9E+09,9E+09,9E+09,9E+09,9E+09,9E+09]],printSpeed,z0,bendedTool\WObj:=wobjpro3;
MoveL [[847.897,325.313,569.01],[0,0.997564,0.069756,0],[0,-1,0,0],[9E+09,9E+09,9E+09,9E+09,9E+09,9E+09]],printSpeed,z0,bendedTool\WObj:=wobjpro3;
MoveL [[846.22,325.215,569.01],[0,0.997564,0.069756,0],[0,-1,0,0],[9E+09,9E+09,9E+09,9E+09,9E+09,9E+09]],printSpeed,z0,bendedTool\WObj:=wobjpro3;
MoveL [[844.547,325.06,569.01],[0,0.997564,0.069756,0],[0,-1,0,0],[9E+09,9E+09,9E+09,9E+09,9E+09,9E+09]],printSpeed,z0,bendedTool\WObj:=wobjpro3;
MoveL [[842.88,324.848,569.01],[0,0.997564,0.069756,0],[0,-1,0,0],[9E+09,9E+09,9E+09,9E+09,9E+09,9E+09]],printSpeed,z0,bendedTool\WObj:=wobjpro3;
MoveL [[841.222,324.581,569.01],[0,0.997564,0.069756,0],[0,-1,0,0],[9E+09,9E+09,9E+09,9E+09,9E+09,9E+09]],printSpeed,z0,bendedTool\WObj:=wobjpro3;
MoveL [[839.573,324.259,569.01],[0,0.997564,0.069756,0],[0,-1,0,0],[9E+09,9E+09,9E+09,9E+09,9E+09,9E+09]],printSpeed,z0,bendedTool\WObj:=wobjpro3;
MoveL [[837.936,323.881,569.01],[0,0.997564,0.069756,0],[0,-1,0,0],[9E+09,9E+09,9E+09,9E+09,9E+09,9E+09]],printSpeed,z0,bendedTool\WObj:=wobjpro3;
MoveL [[836.313,323.449,569.01],[0,0.997564,0.069756,0],[0,-1,0,0],[9E+09,9E+09,9E+09,9E+09,9E+09,9E+09]],printSpeed,z0,bendedTool\WObj:=wobjpro3;
MoveL [[834.705,322.962,569.01],[0,0.997564,0.069756,0],[0,-1,0,0],[9E+09,9E+09,9E+09,9E+09,9E+09,9E+09]],printSpeed,z0,bendedTool\WObj:=wobjpro3;
MoveL [[833.107,322.418,569.01],[0,0.997564,0.069756,0],[0,-1,0,0],[9E+09,9E+09,9E+09,9E+09,9E+09,9E+09]],printSpeed,z0,bendedTool\WObj:=wobjpro3;
MoveL [[831.543,321.828,569.01],[0,0.997564,0.069756,0],[0,-1,0,0],[9E+09,9E+09,9E+09,9E+09,9E+09,9E+09]],printSpeed,z0,bendedTool\WObj:=wobjpro3;
MoveL [[829.992,321.181,569.01],[0,0.997564,0.069756,0],[0,-1,0,0],[9E+09,9E+09,9E+09,9E+09,9E+09,9E+09]],printSpeed,z0,bendedTool\WObj:=wobjpro3;
MoveL [[828.464,320.484,569.01],[0,0.997564,0.069756,0],[0,-1,0,0],[9E+09,9E+09,9E+09,9E+09,9E+09,9E+09]],printSpeed,z0,bendedTool\WObj:=wobjpro3;
MoveL [[826.96,319.735,569.01],[0,0.997564,0.069756,0],[0,-1,0,0],[9E+09,9E+09,9E+09,9E+09,9E+09,9E+09]],printSpeed,z0,bendedTool\WObj:=wobjpro3;
MoveL [[825.483,318.936,569.01],[0,0.997564,0.069756,0],[0,-1,0,0],[9E+09,9E+09,9E+09,9E+09,9E+09,9E+09]],printSpeed,z0,bendedTool\WObj:=wobjpro3;
MoveL [[824.032,318.088,569.01],[0,0.997564,0.069756,0],[0,-1,0,0],[9E+09,9E+09,9E+09,9E+09,9E+09,9E+09]],printSpeed,z0,bendedTool\WObj:=wobjpro3;
MoveL [[822.612,317.191,569.01],[0,0.997564,0.069756,0],[0,-1,0,0],[9E+09,9E+09,9E+09,9E+09,9E+09,9E+09]],printSpeed,z0,bendedTool\WObj:=wobjpro3;
MoveL [[821.222,316.248,569.01],[0,0.997564,0.069756,0],[0,-1,0,0],[9E+09,9E+09,9E+09,9E+09,9E+09,9E+09]],printSpeed,z0,bendedTool\WObj:=wobjpro3;
MoveL [[819.864,315.258,569.01],[0,0.997564,0.069756,0],[0,-1,0,0],[9E+09,9E+09,9E+09,9E+09,9E+09,9E+09]],printSpeed,z0,bendedTool\WObj:=wobjpro3;
MoveL [[818.541,314.223,569.01],[0,0.997564,0.069756,0],[0,-1,0,0],[9E+09,9E+09,9E+09,9E+09,9E+09,9E+09]],printSpeed,z0,bendedTool\WObj:=wobjpro3;
MoveL [[817.253,313.145,569.01],[0,0.997564,0.069756,0],[0,-1,0,0],[9E+09,9E+09,9E+09,9E+09,9E+09,9E+09]],printSpeed,z0,bendedTool\WObj:=wobjpro3;
MoveL [[815.996,312.018,569.01],[0,0.997564,0.069756,0],[0,-1,0,0],[9E+09,9E+09,9E+09,9E+09,9E+09,9E+09]],printSpeed,z0,bendedTool\WObj:=wobjpro3;
MoveL [[814.789,310.861,569.01],[0,0.997564,0.069756,0],[0,-1,0,0],[9E+09,9E+09,9E+09,9E+09,9E+09,9E+09]],printSpeed,z0,bendedTool\WObj:=wobjpro3;
MoveL [[813.617,309.658,569.01],[0,0.997564,0.069756,0],[0,-1,0,0],[9E+09,9E+09,9E+09,9E+09,9E+09,9E+09]],printSpeed,z0,bendedTool\WObj:=wobjpro3;
MoveL [[812.485,308.417,569.01],[0,0.997564,0.069756,0],[0,-1,0,0],[9E+09,9E+09,9E+09,9E+09,9E+09,9E+09]],printSpeed,z0,bendedTool\WObj:=wobjpro3;
MoveL [[811.395,307.138,569.01],[0,0.997564,0.069756,0],[0,-1,0,0],[9E+09,9E+09,9E+09,9E+09,9E+09,9E+09]],printSpeed,z0,bendedTool\WObj:=wobjpro3;
MoveL [[810.35,305.823,569.01],[0,0.997564,0.069756,0],[0,-1,0,0],[9E+09,9E+09,9E+09,9E+09,9E+09,9E+09]],printSpeed,z0,bendedTool\WObj:=wobjpro3;
MoveL [[809.349,304.474,569.01],[0,0.997564,0.069756,0],[0,-1,0,0],[9E+09,9E+09,9E+09,9E+09,9E+09,9E+09]],printSpeed,z0,bendedTool\WObj:=wobjpro3;
MoveL [[808.393,303.092,569.01],[0,0.997564,0.069756,0],[0,-1,0,0],[9E+09,9E+09,9E+09,9E+09,9E+09,9E+09]],printSpeed,z0,bendedTool\WObj:=wobjpro3;
MoveL [[807.485,301.679,569.01],[0,0.997564,0.069756,0],[0,-1,0,0],[9E+09,9E+09,9E+09,9E+09,9E+09,9E+09]],printSpeed,z0,bendedTool\WObj:=wobjpro3;
MoveL [[806.625,300.236,569.01],[0,0.997564,0.069756,0],[0,-1,0,0],[9E+09,9E+09,9E+09,9E+09,9E+09,9E+09]],printSpeed,z0,bendedTool\WObj:=wobjpro3;
MoveL [[805.81,298.757,569.01],[0,0.997564,0.069756,0],[0,-1,0,0],[9E+09,9E+09,9E+09,9E+09,9E+09,9E+09]],printSpeed,z0,bendedTool\WObj:=wobjpro3;
MoveL [[805.052,297.267,569.01],[0,0.997564,0.069756,0],[0,-1,0,0],[9E+09,9E+09,9E+09,9E+09,9E+09,9E+09]],printSpeed,z0,bendedTool\WObj:=wobjpro3;
MoveL [[804.342,295.745,569.01],[0,0.997564,0.069756,0],[0,-1,0,0],[9E+09,9E+09,9E+09,9E+09,9E+09,9E+09]],printSpeed,z0,bendedTool\WObj:=wobjpro3;
MoveL [[803.682,294.2,569.01],[0,0.997564,0.069756,0],[0,-1,0,0],[9E+09,9E+09,9E+09,9E+09,9E+09,9E+09]],printSpeed,z0,bendedTool\WObj:=wobjpro3;
MoveL [[803.076,292.634,569.01],[0,0.997564,0.069756,0],[0,-1,0,0],[9E+09,9E+09,9E+09,9E+09,9E+09,9E+09]],printSpeed,z0,bendedTool\WObj:=wobjpro3;
MoveL [[802.522,291.048,569.01],[0,0.997564,0.069756,0],[0,-1,0,0],[9E+09,9E+09,9E+09,9E+09,9E+09,9E+09]],printSpeed,z0,bendedTool\WObj:=wobjpro3;
MoveL [[802.019,289.436,569.01],[0,0.997564,0.069756,0],[0,-1,0,0],[9E+09,9E+09,9E+09,9E+09,9E+09,9E+09]],printSpeed,z0,bendedTool\WObj:=wobjpro3;
MoveL [[801.575,287.824,569.01],[0,0.997564,0.069756,0],[0,-1,0,0],[9E+09,9E+09,9E+09,9E+09,9E+09,9E+09]],printSpeed,z0,bendedTool\WObj:=wobjpro3;
MoveL [[801.184,286.191,569.01],[0,0.997564,0.069756,0],[0,-1,0,0],[9E+09,9E+09,9E+09,9E+09,9E+09,9E+09]],printSpeed,z0,bendedTool\WObj:=wobjpro3;
MoveL [[800.847,284.545,569.01],[0,0.997564,0.069756,0],[0,-1,0,0],[9E+09,9E+09,9E+09,9E+09,9E+09,9E+09]],printSpeed,z0,bendedTool\WObj:=wobjpro3;
MoveL [[800.566,282.889,569.01],[0,0.997564,0.069756,0],[0,-1,0,0],[9E+09,9E+09,9E+09,9E+09,9E+09,9E+09]],printSpeed,z0,bendedTool\WObj:=wobjpro3;
MoveL [[800.34,281.215,569.01],[0,0.997564,0.069756,0],[0,-1,0,0],[9E+09,9E+09,9E+09,9E+09,9E+09,9E+09]],printSpeed,z0,bendedTool\WObj:=wobjpro3;
MoveL [[800.172,279.552,569.01],[0,0.997564,0.069756,0],[0,-1,0,0],[9E+09,9E+09,9E+09,9E+09,9E+09,9E+09]],printSpeed,z0,bendedTool\WObj:=wobjpro3;
MoveL [[800.059,277.876,569.01],[0,0.997564,0.069756,0],[0,-1,0,0],[9E+09,9E+09,9E+09,9E+09,9E+09,9E+09]],printSpeed,z0,bendedTool\WObj:=wobjpro3;
MoveL [[800.003,276.197,569.01],[0,0.997564,0.069756,0],[0,-1,0,0],[9E+09,9E+09,9E+09,9E+09,9E+09,9E+09]],printSpeed,z0,bendedTool\WObj:=wobjpro3;
MoveL [[800.003,274.517,569.01],[0,0.997564,0.069756,0],[0,-1,0,0],[9E+09,9E+09,9E+09,9E+09,9E+09,9E+09]],printSpeed,z0,bendedTool\WObj:=wobjpro3;
MoveL [[800.059,272.838,569.01],[0,0.997564,0.069756,0],[0,-1,0,0],[9E+09,9E+09,9E+09,9E+09,9E+09,9E+09]],printSpeed,z0,bendedTool\WObj:=wobjpro3;
MoveL [[800.172,271.162,569.01],[0,0.997564,0.069756,0],[0,-1,0,0],[9E+09,9E+09,9E+09,9E+09,9E+09,9E+09]],printSpeed,z0,bendedTool\WObj:=wobjpro3;
MoveL [[800.341,269.491,569.01],[0,0.997564,0.069756,0],[0,-1,0,0],[9E+09,9E+09,9E+09,9E+09,9E+09,9E+09]],printSpeed,z0,bendedTool\WObj:=wobjpro3;
MoveL [[800.566,267.826,569.01],[0,0.997564,0.069756,0],[0,-1,0,0],[9E+09,9E+09,9E+09,9E+09,9E+09,9E+09]],printSpeed,z0,bendedTool\WObj:=wobjpro3;
MoveL [[800.847,266.17,569.01],[0,0.997564,0.069756,0],[0,-1,0,0],[9E+09,9E+09,9E+09,9E+09,9E+09,9E+09]],printSpeed,z0,bendedTool\WObj:=wobjpro3;
MoveL [[801.184,264.524,569.01],[0,0.997564,0.069756,0],[0,-1,0,0],[9E+09,9E+09,9E+09,9E+09,9E+09,9E+09]],printSpeed,z0,bendedTool\WObj:=wobjpro3;
MoveL [[801.575,262.89,569.01],[0,0.997564,0.069756,0],[0,-1,0,0],[9E+09,9E+09,9E+09,9E+09,9E+09,9E+09]],printSpeed,fine,bendedTool\WObj:=wobjpro3;
stopContinuousWeld \delay:=delayClosedStop_0;
Tperase;
TPWrite "PRT0 is done printing";
MoveL [[801.575,262.89,669.01],[0,0.997564,0.069756,0],[0,-1,0,0],[9E+09,9E+09,9E+09,9E+09,9E+09,9E+09]],moveSpeed,z0,bendedTool\WObj:=wobjpro3;
tidyUp;
ENDPROC

PROC r_cutwire()

ENDPROC
PROC startcontinuousweld()

ENDPROC
PROC tidyUp()

ENDPROC
PROC stopContinuousWeld(\num delay)

ENDPROC
PROC serch_height(num ofx, num ofy, robtarget target, inout num zval)

ENDPROC
PROC waitInterpass(bool useTempSensor, num wTime)

ENDPROC

ENDMODULE
